LIN {X 0,Y 573.095,Z 768.426,A -85,B 0,C 180,E1 -2257.752,E2 -2257.752} C_VEL
LIN {X 0,Y 573.136,Z 760.652,A -85,B 0,C 180,E1 -2259.172,E2 -2259.172} C_VEL
LIN {X 0,Y 573.27,Z 752.373,A -85,B 0,C 180,E1 -2260.417,E2 -2260.417} C_VEL
LIN {X 0,Y 573.384,Z 742.397,A -85,B 0,C 180,E1 -2261.667,E2 -2261.667} C_VEL
LIN {X 0,Y 573.567,Z 732.195,A -85,B 0,C 180,E1 -2262.741,E2 -2262.741} C_VEL
LIN {X 0,Y 573.742,Z 720.027,A -85,B 0,C 180,E1 -2263.819,E2 -2263.819} C_VEL
LIN {X 0,Y 573.959,Z 706.912,A -85,B 0,C 180,E1 -2264.78,E2 -2264.78} C_VEL
LIN {X 0,Y 574.138,Z 692.882,A -85,B 0,C 180,E1 -2265.622,E2 -2265.622} C_VEL
LIN {X 0,Y 574.337,Z 678.815,A -85,B 0,C 180,E1 -2266.3,E2 -2266.3} C_VEL
LIN {X 0,Y 574.521,Z 664.326,A -85,B 0,C 180,E1 -2266.843,E2 -2266.843} C_VEL
LIN {X 0,Y 574.696,Z 648.452,A -85,B 0,C 180,E1 -2267.274,E2 -2267.274} C_VEL
LIN {X 0,Y 574.79,Z 632.509,A -85,B 0,C 180,E1 -2267.547,E2 -2267.547} C_VEL
LIN {X 0,Y 575.114,Z 478.185,A -85,B 0,C 180,E1 -2269.528,E2 -2269.528} C_VEL
LIN {X 0,Y 574.295,Z 472.988,A -85,B 0,C 180,E1 -2269.647,E2 -2269.647} C_VEL
LIN {X 0,Y 574.659,Z 443.059,A -85,B 0,C 180,E1 -2272.468,E2 -2272.468} C_VEL
LIN {X 0,Y 575.111,Z 413.325,A -85,B 0,C 180,E1 -2275.321,E2 -2275.321} C_VEL
LIN {X 0,Y 575.49,Z 387.313,A -85,B 0,C 180,E1 -2277.839,E2 -2277.839} C_VEL
LIN {X 0,Y 575.461,Z 368.493,A -85,B 0,C 180,E1 -2279.623,E2 -2279.623} C_VEL
LIN {X 0,Y 573.25,Z 359.705,A -85,B 0,C 180,E1 -2280.582,E2 -2280.582} C_VEL
LIN {X 0,Y 573.235,Z 359.704,A -85,B 0,C 180,E1 -2283.52,E2 -2283.52} C_VEL
LIN {X 0,Y 573.175,Z 359.715,A -85,B 0,C 180,E1 -2286.053,E2 -2286.053} C_VEL
LIN {X 0,Y 573.22,Z 359.704,A -85,B 0,C 180,E1 -2288.702,E2 -2288.702} C_VEL
LIN {X 0,Y 573.191,Z 359.706,A -85,B 0,C 180,E1 -2291.459,E2 -2291.459} C_VEL
LIN {X 0,Y 573.203,Z 359.709,A -85,B 0,C 180,E1 -2294.335,E2 -2294.335} C_VEL
LIN {X 0,Y 573.197,Z 359.704,A -85,B 0,C 180,E1 -2297.361,E2 -2297.361} C_VEL
LIN {X 0,Y 573.217,Z 359.708,A -85,B 0,C 180,E1 -2300.391,E2 -2300.391} C_VEL
LIN {X 0,Y 573.201,Z 359.704,A -85,B 0,C 180,E1 -2303.074,E2 -2303.074} C_VEL
LIN {X 0,Y 573.228,Z 359.702,A -85,B 0,C 180,E1 -2305.669,E2 -2305.669} C_VEL
LIN {X 0,Y 573.208,Z 359.712,A -85,B 0,C 180,E1 -2308.183,E2 -2308.183} C_VEL
LIN {X 0,Y 573.205,Z 359.709,A -85,B 0,C 180,E1 -2310.631,E2 -2310.631} C_VEL
LIN {X 0,Y 573.189,Z 359.706,A -85,B 0,C 180,E1 -2313.514,E2 -2313.514} C_VEL
LIN {X 0,Y 573.178,Z 359.713,A -85,B 0,C 180,E1 -2316.132,E2 -2316.132} C_VEL
LIN {X 0,Y 573.201,Z 359.704,A -85,B 0,C 180,E1 -2319.172,E2 -2319.172} C_VEL
LIN {X 0,Y 573.174,Z 359.707,A -85,B 0,C 180,E1 -2321.41,E2 -2321.41} C_VEL
LIN {X 0,Y 573.186,Z 359.715,A -85,B 0,C 180,E1 -2324.351,E2 -2324.351} C_VEL
LIN {X 0,Y 573.173,Z 359.717,A -85,B 0,C 180,E1 -2326.528,E2 -2326.528} C_VEL
LIN {X 0,Y 573.221,Z 359.701,A -85,B 0,C 180,E1 -2329.403,E2 -2329.403} C_VEL
LIN {X 0,Y 573.219,Z 359.708,A -85,B 0,C 180,E1 -2332.249,E2 -2332.249} C_VEL
LIN {X 0,Y 573.262,Z 359.698,A -85,B 0,C 180,E1 -2335.077,E2 -2335.077} C_VEL
LIN {X 0,Y 573.269,Z 359.695,A -85,B 0,C 180,E1 -2337.892,E2 -2337.892} C_VEL
LIN {X 0,Y 573.317,Z 359.697,A -85,B 0,C 180,E1 -2340.703,E2 -2340.703} C_VEL
LIN {X 0,Y 573.283,Z 359.7,A -85,B 0,C 180,E1 -2342.811,E2 -2342.811} C_VEL
LIN {X 0,Y 573.245,Z 359.696,A -85,B 0,C 180,E1 -2345.629,E2 -2345.629} C_VEL
LIN {X 0,Y 573.198,Z 359.7,A -85,B 0,C 180,E1 -2347.751,E2 -2347.751} C_VEL
LIN {X 0,Y 573.23,Z 359.709,A -85,B 0,C 180,E1 -2350.598,E2 -2350.598} C_VEL
LIN {X 0,Y 573.196,Z 359.702,A -85,B 0,C 180,E1 -2353.472,E2 -2353.472} C_VEL
LIN {X 0,Y 573.206,Z 359.701,A -85,B 0,C 180,E1 -2355.649,E2 -2355.649} C_VEL
LIN {X 0,Y 573.207,Z 359.703,A -85,B 0,C 180,E1 -2357.85,E2 -2357.85} C_VEL
LIN {X 0,Y 573.222,Z 359.7,A -85,B 0,C 180,E1 -2360.078,E2 -2360.078} C_VEL
LIN {X 0,Y 573.208,Z 359.704,A -85,B 0,C 180,E1 -2362.339,E2 -2362.339} C_VEL
LIN {X 0,Y 573.193,Z 359.709,A -85,B 0,C 180,E1 -2364.401,E2 -2364.401} C_VEL
LIN {X 0,Y 572.552,Z 359.795,A -85,B 0,C 180,E1 -2364.987,E2 -2364.987} C_VEL
LIN {X 0,Y 569.7,Z 360.151,A -85,B 0,C 180,E1 -2365.939,E2 -2365.939} C_VEL
LIN {X 0,Y 567.274,Z 360.449,A -85,B 0,C 180,E1 -2366.705,E2 -2366.705} C_VEL
LIN {X 0,Y 566.232,Z 360.574,A -85,B 0,C 180,E1 -2367.296,E2 -2367.296} C_VEL
LIN {X 0,Y 566.147,Z 360.583,A -85,B 0,C 180,E1 -2367.496,E2 -2367.496} C_VEL
LIN {X 0,Y 566.158,Z 360.582,A -85,B 0,C 180,E1 -2369.772,E2 -2369.772} C_VEL
LIN {X 0,Y 566.188,Z 360.578,A -85,B 0,C 180,E1 -2372.43,E2 -2372.43} C_VEL
LIN {X 0,Y 566.168,Z 360.588,A -85,B 0,C 180,E1 -2374.99,E2 -2374.99} C_VEL
LIN {X 0,Y 566.184,Z 360.58,A -85,B 0,C 180,E1 -2377.462,E2 -2377.462} C_VEL
LIN {X 0,Y 566.196,Z 360.577,A -85,B 0,C 180,E1 -2380.2,E2 -2380.2} C_VEL
LIN {X 0,Y 566.176,Z 360.586,A -85,B 0,C 180,E1 -2383.057,E2 -2383.057} C_VEL
LIN {X 0,Y 566.185,Z 360.578,A -85,B 0,C 180,E1 -2386.051,E2 -2386.051} C_VEL
LIN {X 0,Y 566.195,Z 360.583,A -85,B 0,C 180,E1 -2389.216,E2 -2389.216} C_VEL
LIN {X 0,Y 566.173,Z 360.581,A -85,B 0,C 180,E1 -2391.637,E2 -2391.637} C_VEL
LIN {X 0,Y 566.138,Z 360.584,A -85,B 0,C 180,E1 -2394.307,E2 -2394.307} C_VEL
LIN {X 0,Y 566.191,Z 360.585,A -85,B 0,C 180,E1 -2396.897,E2 -2396.897} C_VEL
LIN {X 0,Y 566.16,Z 360.588,A -85,B 0,C 180,E1 -2399.407,E2 -2399.407} C_VEL
LIN {X 0,Y 566.169,Z 360.587,A -85,B 0,C 180,E1 -2401.612,E2 -2401.612} C_VEL
LIN {X 0,Y 568.353,Z 366.669,A -85,B 0,C 180,E1 -2401.781,E2 -2401.781} C_VEL
LIN {X 0,Y 567.975,Z 490.989,A -85,B 0,C 180,E1 -2403.409,E2 -2403.409} C_VEL
LIN {X 0,Y 567.841,Z 506.693,A -85,B 0,C 180,E1 -2403.764,E2 -2403.764} C_VEL
LIN {X 0,Y 567.638,Z 522.129,A -85,B 0,C 180,E1 -2404.272,E2 -2404.272} C_VEL
LIN {X 0,Y 567.384,Z 536.347,A -85,B 0,C 180,E1 -2404.89,E2 -2404.89} C_VEL
LIN {X 0,Y 567.131,Z 550.503,A -85,B 0,C 180,E1 -2405.668,E2 -2405.668} C_VEL
LIN {X 0,Y 566.889,Z 563.595,A -85,B 0,C 180,E1 -2406.552,E2 -2406.552} C_VEL
LIN {X 0,Y 566.633,Z 576.205,A -85,B 0,C 180,E1 -2407.581,E2 -2407.581} C_VEL
LIN {X 0,Y 566.434,Z 587.684,A -85,B 0,C 180,E1 -2408.706,E2 -2408.706} C_VEL
LIN {X 0,Y 566.289,Z 597.552,A -85,B 0,C 180,E1 -2409.856,E2 -2409.856} C_VEL
LIN {X 0,Y 566.118,Z 606.994,A -85,B 0,C 180,E1 -2411.17,E2 -2411.17} C_VEL
LIN {X 0,Y 566.04,Z 614.754,A -85,B 0,C 180,E1 -2412.478,E2 -2412.478} C_VEL
LIN {X 0,Y 565.979,Z 621.094,A -85,B 0,C 180,E1 -2413.777,E2 -2413.777} C_VEL
LIN {X 0,Y 565.932,Z 626.848,A -85,B 0,C 180,E1 -2415.252,E2 -2415.252} C_VEL
LIN {X 0,Y 565.884,Z 630.24,A -85,B 0,C 180,E1 -2416.352,E2 -2416.352} C_VEL
LIN {X 0,Y 565.865,Z 633.545,A -85,B 0,C 180,E1 -2417.812,E2 -2417.812} C_VEL
LIN {X 0,Y 565.89,Z 635.583,A -85,B 0,C 180,E1 -2419.264,E2 -2419.264} C_VEL
LIN {X 0,Y 565.822,Z 636.432,A -85,B 0,C 180,E1 -2420.708,E2 -2420.708} C_VEL
LIN {X 0,Y 565.876,Z 636.125,A -85,B 0,C 180,E1 -2422.148,E2 -2422.148} C_VEL
LIN {X 0,Y 565.897,Z 634.669,A -85,B 0,C 180,E1 -2423.583,E2 -2423.583} C_VEL
LIN {X 0,Y 565.855,Z 632.049,A -85,B 0,C 180,E1 -2425.013,E2 -2425.013} C_VEL
LIN {X 0,Y 565.948,Z 628.168,A -85,B 0,C 180,E1 -2426.441,E2 -2426.441} C_VEL
LIN {X 0,Y 565.905,Z 623.007,A -85,B 0,C 180,E1 -2427.865,E2 -2427.865} C_VEL
LIN {X 0,Y 566.023,Z 616.441,A -85,B 0,C 180,E1 -2429.289,E2 -2429.289} C_VEL
LIN {X 0,Y 566.103,Z 609.405,A -85,B 0,C 180,E1 -2430.534,E2 -2430.534} C_VEL
LIN {X 0,Y 566.216,Z 600.993,A -85,B 0,C 180,E1 -2431.778,E2 -2431.778} C_VEL
LIN {X 0,Y 566.393,Z 590.924,A -85,B 0,C 180,E1 -2433.023,E2 -2433.023} C_VEL
LIN {X 0,Y 566.631,Z 580.682,A -85,B 0,C 180,E1 -2434.09,E2 -2434.09} C_VEL
LIN {X 0,Y 566.799,Z 568.495,A -85,B 0,C 180,E1 -2435.158,E2 -2435.158} C_VEL
LIN {X 0,Y 567.019,Z 556.344,A -85,B 0,C 180,E1 -2436.048,E2 -2436.048} C_VEL
LIN {X 0,Y 567.283,Z 543.123,A -85,B 0,C 180,E1 -2436.849,E2 -2436.849} C_VEL
LIN {X 0,Y 567.537,Z 528.88,A -85,B 0,C 180,E1 -2437.543,E2 -2437.543} C_VEL
LIN {X 0,Y 567.774,Z 514.325,A -85,B 0,C 180,E1 -2438.094,E2 -2438.094} C_VEL
LIN {X 0,Y 567.889,Z 499.072,A -85,B 0,C 180,E1 -2438.518,E2 -2438.518} C_VEL
LIN {X 0,Y 567.973,Z 484.215,A -85,B 0,C 180,E1 -2438.786,E2 -2438.786} C_VEL
LIN {X 0,Y 568.274,Z 366.453,A -85,B 0,C 180,E1 -2440.315,E2 -2440.315} C_VEL
LIN {X 0,Y 566.187,Z 360.585,A -85,B 0,C 180,E1 -2440.482,E2 -2440.482} C_VEL
LIN {X 0,Y 566.145,Z 360.593,A -85,B 0,C 180,E1 -2442.912,E2 -2442.912} C_VEL
LIN {X 0,Y 566.155,Z 360.59,A -85,B 0,C 180,E1 -2445.111,E2 -2445.111} C_VEL
LIN {X 0,Y 566.161,Z 360.581,A -85,B 0,C 180,E1 -2448.079,E2 -2448.079} C_VEL
LIN {X 0,Y 566.15,Z 360.584,A -85,B 0,C 180,E1 -2450.339,E2 -2450.339} C_VEL
LIN {X 0,Y 566.131,Z 360.589,A -85,B 0,C 180,E1 -2452.633,E2 -2452.633} C_VEL
LIN {X 0,Y 566.141,Z 360.593,A -85,B 0,C 180,E1 -2455.012,E2 -2455.012} C_VEL
LIN {X 0,Y 566.158,Z 360.587,A -85,B 0,C 180,E1 -2457.341,E2 -2457.341} C_VEL
LIN {X 0,Y 566.143,Z 360.581,A -85,B 0,C 180,E1 -2459.772,E2 -2459.772} C_VEL
LIN {X 0,Y 566.169,Z 360.581,A -85,B 0,C 180,E1 -2462.424,E2 -2462.424} C_VEL
LIN {X 0,Y 566.154,Z 360.589,A -85,B 0,C 180,E1 -2464.985,E2 -2464.985} C_VEL
LIN {X 0,Y 566.184,Z 360.583,A -85,B 0,C 180,E1 -2467.461,E2 -2467.461} C_VEL
LIN {X 0,Y 566.16,Z 360.58,A -85,B 0,C 180,E1 -2470.202,E2 -2470.202} C_VEL
LIN {X 0,Y 566.139,Z 360.592,A -85,B 0,C 180,E1 -2473.059,E2 -2473.059} C_VEL
LIN {X 0,Y 566.147,Z 360.583,A -85,B 0,C 180,E1 -2476.053,E2 -2476.053} C_VEL
LIN {X 0,Y 566.165,Z 360.59,A -85,B 0,C 180,E1 -2479.218,E2 -2479.218} C_VEL
LIN {X 0,Y 566.138,Z 360.587,A -85,B 0,C 180,E1 -2481.633,E2 -2481.633} C_VEL
LIN {X 0,Y 566.133,Z 360.584,A -85,B 0,C 180,E1 -2484.305,E2 -2484.305} C_VEL
LIN {X 0,Y 566.154,Z 360.584,A -85,B 0,C 180,E1 -2486.893,E2 -2486.893} C_VEL
LIN {X 0,Y 566.141,Z 360.591,A -85,B 0,C 180,E1 -2489.405,E2 -2489.405} C_VEL
LIN {X 0,Y 566.138,Z 360.586,A -85,B 0,C 180,E1 -2491.853,E2 -2491.853} C_VEL
LIN {X 0,Y 566.158,Z 360.581,A -85,B 0,C 180,E1 -2494.248,E2 -2494.248} C_VEL
LIN {X 0,Y 566.151,Z 360.592,A -85,B 0,C 180,E1 -2497.367,E2 -2497.367} C_VEL
LIN {X 0,Y 566.189,Z 360.582,A -85,B 0,C 180,E1 -2499.662,E2 -2499.662} C_VEL
LIN {X 0,Y 566.156,Z 360.583,A -85,B 0,C 180,E1 -2501.92,E2 -2501.92} C_VEL
LIN {X 0,Y 566.172,Z 360.582,A -85,B 0,C 180,E1 -2504.89,E2 -2504.89} C_VEL
LIN {X 0,Y 566.165,Z 360.578,A -85,B 0,C 180,E1 -2507.817,E2 -2507.817} C_VEL
LIN {X 0,Y 566.126,Z 360.582,A -85,B 0,C 180,E1 -2509.991,E2 -2509.991} C_VEL
LIN {X 0,Y 566.168,Z 360.579,A -85,B 0,C 180,E1 -2512.152,E2 -2512.152} C_VEL
LIN {X 0,Y 566.255,Z 360.572,A -85,B 0,C 180,E1 -2515.016,E2 -2515.016} C_VEL
LIN {X 0,Y 566.248,Z 360.573,A -85,B 0,C 180,E1 -2517.866,E2 -2517.866} C_VEL
LIN {X 0,Y 566.255,Z 360.572,A -85,B 0,C 180,E1 -2520,E2 -2520} C_VEL
LIN {X 0,Y 566.233,Z 360.572,A -85,B 0,C 180,E1 -2522.846,E2 -2522.846} C_VEL
LIN {X 0,Y 566.223,Z 360.581,A -85,B 0,C 180,E1 -2525.698,E2 -2525.698} C_VEL
LIN {X 0,Y 566.165,Z 360.579,A -85,B 0,C 180,E1 -2528.566,E2 -2528.566} C_VEL
LIN {X 0,Y 566.226,Z 360.58,A -85,B 0,C 180,E1 -2531.454,E2 -2531.454} C_VEL
LIN {X 0,Y 566.191,Z 360.576,A -85,B 0,C 180,E1 -2534.494,E2 -2534.494} C_VEL
LIN {X 0,Y 566.146,Z 360.588,A -85,B 0,C 180,E1 -2537.333,E2 -2537.333} C_VEL
LIN {X 0,Y 566.163,Z 360.588,A -85,B 0,C 180,E1 -2539.582,E2 -2539.582} C_VEL
LIN {X 0,Y 566.135,Z 360.59,A -85,B 0,C 180,E1 -2541.865,E2 -2541.865} C_VEL
LIN {X 0,Y 566.183,Z 360.579,A -85,B 0,C 180,E1 -2544.963,E2 -2544.963} C_VEL
LIN {X 0,Y 566.148,Z 360.586,A -85,B 0,C 180,E1 -2547.342,E2 -2547.342} C_VEL
LIN {X 0,Y 566.149,Z 360.592,A -85,B 0,C 180,E1 -2549.772,E2 -2549.772} C_VEL
LIN {X 0,Y 566.166,Z 360.58,A -85,B 0,C 180,E1 -2552.426,E2 -2552.426} C_VEL
LIN {X 0,Y 566.153,Z 360.581,A -85,B 0,C 180,E1 -2554.987,E2 -2554.987} C_VEL
LIN {X 0,Y 566.173,Z 360.584,A -85,B 0,C 180,E1 -2557.463,E2 -2557.463} C_VEL
LIN {X 0,Y 566.195,Z 360.581,A -85,B 0,C 180,E1 -2560.2,E2 -2560.2} C_VEL
LIN {X 0,Y 566.134,Z 360.584,A -85,B 0,C 180,E1 -2563.06,E2 -2563.06} C_VEL
LIN {X 0,Y 566.147,Z 360.59,A -85,B 0,C 180,E1 -2566.054,E2 -2566.054} C_VEL
LIN {X 0,Y 566.132,Z 360.582,A -85,B 0,C 180,E1 -2568.858,E2 -2568.858} C_VEL
LIN {X 0,Y 566.167,Z 360.586,A -85,B 0,C 180,E1 -2571.636,E2 -2571.636} C_VEL
LIN {X 0,Y 566.131,Z 360.59,A -85,B 0,C 180,E1 -2574.306,E2 -2574.306} C_VEL
LIN {X 0,Y 566.158,Z 360.584,A -85,B 0,C 180,E1 -2576.894,E2 -2576.894} C_VEL
LIN {X 0,Y 566.183,Z 360.71,A -85,B 0,C 180,E1 -2579.186,E2 -2579.186} C_VEL
LIN {X 0,Y 568.608,Z 369.797,A -85,B 0,C 180,E1 -2580.186,E2 -2580.186} C_VEL
LIN {X 0,Y 568.694,Z 381.61,A -85,B 0,C 180,E1 -2581.333,E2 -2581.333} C_VEL
LIN {X 0,Y 568.501,Z 408.247,A -85,B 0,C 180,E1 -2583.871,E2 -2583.871} C_VEL
LIN {X 0,Y 568.018,Z 435.853,A -85,B 0,C 180,E1 -2586.554,E2 -2586.554} C_VEL
LIN {X 0,Y 567.548,Z 464.858,A -85,B 0,C 180,E1 -2589.334,E2 -2589.334} C_VEL
LIN {X 0,Y 567.46,Z 473.303,A -85,B 0,C 180,E1 -2590.133,E2 -2590.133} C_VEL
LIN {X 0,Y 568.498,Z 480.342,A -85,B 0,C 180,E1 -2590.264,E2 -2590.264} C_VEL
LIN {X 0,Y 567.995,Z 640.714,A -85,B 0,C 180,E1 -2592.36,E2 -2592.36} C_VEL
LIN {X 0,Y 567.839,Z 656.165,A -85,B 0,C 180,E1 -2592.705,E2 -2592.705} C_VEL
LIN {X 0,Y 567.658,Z 670.801,A -85,B 0,C 180,E1 -2593.178,E2 -2593.178} C_VEL
LIN {X 0,Y 567.491,Z 683.806,A -85,B 0,C 180,E1 -2593.728,E2 -2593.728} C_VEL
LIN {X 0,Y 567.175,Z 697.681,A -85,B 0,C 180,E1 -2594.457,E2 -2594.457} C_VEL
LIN {X 0,Y 566.935,Z 711.501,A -85,B 0,C 180,E1 -2595.358,E2 -2595.358} C_VEL
LIN {X 0,Y 566.672,Z 724.291,A -85,B 0,C 180,E1 -2596.371,E2 -2596.371} C_VEL
LIN {X 0,Y 566.491,Z 735.749,A -85,B 0,C 180,E1 -2597.461,E2 -2597.461} C_VEL
LIN {X 0,Y 566.268,Z 746.312,A -85,B 0,C 180,E1 -2598.659,E2 -2598.659} C_VEL
LIN {X 0,Y 566.208,Z 754.857,A -85,B 0,C 180,E1 -2599.812,E2 -2599.812} C_VEL
LIN {X 0,Y 566.057,Z 762.733,A -85,B 0,C 180,E1 -2601.072,E2 -2601.072} C_VEL
LIN {X 0,Y 565.997,Z 770.089,A -85,B 0,C 180,E1 -2602.508,E2 -2602.508} C_VEL
LIN {X 0,Y 565.956,Z 775.922,A -85,B 0,C 180,E1 -2603.941,E2 -2603.941} C_VEL
LIN {X 0,Y 565.866,Z 779.385,A -85,B 0,C 180,E1 -2605.012,E2 -2605.012} C_VEL
LIN {X 0,Y 565.909,Z 782.889,A -85,B 0,C 180,E1 -2606.44,E2 -2606.44} C_VEL
LIN {X 0,Y 565.836,Z 785.192,A -85,B 0,C 180,E1 -2607.864,E2 -2607.864} C_VEL
LIN {X 0,Y 565.838,Z 786.349,A -85,B 0,C 180,E1 -2609.288,E2 -2609.288} C_VEL
LIN {X 0,Y 565.838,Z 786.349,A -85,B 0,C 180,E1 -2610.711,E2 -2610.711} C_VEL
LIN {X 0,Y 565.836,Z 785.191,A -85,B 0,C 180,E1 -2612.135,E2 -2612.135} C_VEL
LIN {X 0,Y 565.909,Z 782.888,A -85,B 0,C 180,E1 -2613.56,E2 -2613.56} C_VEL
LIN {X 0,Y 565.866,Z 779.387,A -85,B 0,C 180,E1 -2614.987,E2 -2614.987} C_VEL
LIN {X 0,Y 565.956,Z 775.926,A -85,B 0,C 180,E1 -2616.059,E2 -2616.059} C_VEL
LIN {X 0,Y 565.999,Z 770.09,A -85,B 0,C 180,E1 -2617.491,E2 -2617.491} C_VEL
LIN {X 0,Y 566.057,Z 762.733,A -85,B 0,C 180,E1 -2618.928,E2 -2618.928} C_VEL
LIN {X 0,Y 566.208,Z 754.86,A -85,B 0,C 180,E1 -2620.187,E2 -2620.187} C_VEL
LIN {X 0,Y 566.307,Z 745.395,A -85,B 0,C 180,E1 -2621.452,E2 -2621.452} C_VEL
LIN {X 0,Y 566.491,Z 735.754,A -85,B 0,C 180,E1 -2622.539,E2 -2622.539} C_VEL
LIN {X 0,Y 566.671,Z 724.301,A -85,B 0,C 180,E1 -2623.629,E2 -2623.629} C_VEL
LIN {X 0,Y 566.926,Z 711.684,A -85,B 0,C 180,E1 -2624.63,E2 -2624.63} C_VEL
LIN {X 0,Y 567.15,Z 699.255,A -85,B 0,C 180,E1 -2625.451,E2 -2625.451} C_VEL
LIN {X 0,Y 567.418,Z 685.782,A -85,B 0,C 180,E1 -2626.181,E2 -2626.181} C_VEL
LIN {X 0,Y 567.606,Z 672.065,A -85,B 0,C 180,E1 -2626.777,E2 -2626.777} C_VEL
LIN {X 0,Y 567.845,Z 656.743,A -85,B 0,C 180,E1 -2627.279,E2 -2627.279} C_VEL
LIN {X 0,Y 567.978,Z 641.336,A -85,B 0,C 180,E1 -2627.629,E2 -2627.629} C_VEL
LIN {X 0,Y 568.451,Z 479.257,A -85,B 0,C 180,E1 -2629.752,E2 -2629.752} C_VEL
LIN {X 0,Y 567.456,Z 473.137,A -85,B 0,C 180,E1 -2629.879,E2 -2629.879} C_VEL
LIN {X 0,Y 567.9,Z 443.059,A -85,B 0,C 180,E1 -2632.75,E2 -2632.75} C_VEL
LIN {X 0,Y 568.442,Z 413.325,A -85,B 0,C 180,E1 -2635.64,E2 -2635.64} C_VEL
LIN {X 0,Y 568.649,Z 384.809,A -85,B 0,C 180,E1 -2638.347,E2 -2638.347} C_VEL
LIN {X 0,Y 568.585,Z 369.664,A -85,B 0,C 180,E1 -2639.805,E2 -2639.805} C_VEL
LIN {X 0,Y 566.189,Z 360.584,A -85,B 0,C 180,E1 -2640.814,E2 -2640.814} C_VEL
LIN {X 0,Y 566.188,Z 360.58,A -85,B 0,C 180,E1 -2643.103,E2 -2643.103} C_VEL
LIN {X 0,Y 566.129,Z 360.59,A -85,B 0,C 180,E1 -2645.693,E2 -2645.693} C_VEL
LIN {X 0,Y 566.191,Z 360.581,A -85,B 0,C 180,E1 -2648.556,E2 -2648.556} C_VEL
LIN {X 0,Y 566.145,Z 360.583,A -85,B 0,C 180,E1 -2651.141,E2 -2651.141} C_VEL
LIN {X 0,Y 566.144,Z 360.59,A -85,B 0,C 180,E1 -2653.946,E2 -2653.946} C_VEL
LIN {X 0,Y 566.135,Z 360.584,A -85,B 0,C 180,E1 -2657.088,E2 -2657.088} C_VEL
LIN {X 0,Y 566.194,Z 360.584,A -85,B 0,C 180,E1 -2660.315,E2 -2660.315} C_VEL
LIN {X 0,Y 566.171,Z 360.584,A -85,B 0,C 180,E1 -2662.601,E2 -2662.601} C_VEL
LIN {X 0,Y 566.166,Z 360.581,A -85,B 0,C 180,E1 -2665.179,E2 -2665.179} C_VEL
LIN {X 0,Y 566.193,Z 360.579,A -85,B 0,C 180,E1 -2667.741,E2 -2667.741} C_VEL
LIN {X 0,Y 566.143,Z 360.593,A -85,B 0,C 180,E1 -2670.336,E2 -2670.336} C_VEL
LIN {X 0,Y 566.164,Z 360.581,A -85,B 0,C 180,E1 -2673.456,E2 -2673.456} C_VEL
LIN {X 0,Y 566.14,Z 360.586,A -85,B 0,C 180,E1 -2675.817,E2 -2675.817} C_VEL
LIN {X 0,Y 566.166,Z 360.582,A -85,B 0,C 180,E1 -2678.901,E2 -2678.901} C_VEL
LIN {X 0,Y 566.151,Z 360.583,A -85,B 0,C 180,E1 -2681.171,E2 -2681.171} C_VEL
LIN {X 0,Y 566.153,Z 360.587,A -85,B 0,C 180,E1 -2684.151,E2 -2684.151} C_VEL
LIN {X 0,Y 566.139,Z 360.592,A -85,B 0,C 180,E1 -2686.358,E2 -2686.358} C_VEL
LIN {X 0,Y 566.2,Z 360.576,A -85,B 0,C 180,E1 -2689.27,E2 -2689.27} C_VEL
LIN {X 0,Y 566.182,Z 360.583,A -85,B 0,C 180,E1 -2692.152,E2 -2692.152} C_VEL
LIN {X 0,Y 566.238,Z 360.574,A -85,B 0,C 180,E1 -2695.016,E2 -2695.016} C_VEL
LIN {X 0,Y 566.242,Z 360.57,A -85,B 0,C 180,E1 -2697.866,E2 -2697.866} C_VEL
LIN {X 0,Y 566.286,Z 360.572,A -85,B 0,C 180,E1 -2700.711,E2 -2700.711} C_VEL
LIN {X 0,Y 566.247,Z 360.576,A -85,B 0,C 180,E1 -2702.846,E2 -2702.846} C_VEL
LIN {X 0,Y 566.215,Z 360.571,A -85,B 0,C 180,E1 -2705.699,E2 -2705.699} C_VEL
LIN {X 0,Y 566.169,Z 360.576,A -85,B 0,C 180,E1 -2707.848,E2 -2707.848} C_VEL
LIN {X 0,Y 566.207,Z 360.584,A -85,B 0,C 180,E1 -2710.731,E2 -2710.731} C_VEL
LIN {X 0,Y 566.162,Z 360.577,A -85,B 0,C 180,E1 -2713.642,E2 -2713.642} C_VEL
LIN {X 0,Y 566.192,Z 360.583,A -85,B 0,C 180,E1 -2716.589,E2 -2716.589} C_VEL
LIN {X 0,Y 566.186,Z 360.576,A -85,B 0,C 180,E1 -2719.582,E2 -2719.582} C_VEL
LIN {X 0,Y 566.172,Z 360.577,A -85,B 0,C 180,E1 -2721.864,E2 -2721.864} C_VEL
LIN {X 0,Y 566.165,Z 360.585,A -85,B 0,C 180,E1 -2725.022,E2 -2725.022} C_VEL
LIN {X 0,Y 566.147,Z 360.583,A -85,B 0,C 180,E1 -2727.496,E2 -2727.496} C_VEL
LIN {X 0,Y 565.48,Z 360.666,A -85,B 0,C 180,E1 -2728.09,E2 -2728.09} C_VEL
LIN {X 0,Y 562.624,Z 361.029,A -85,B 0,C 180,E1 -2729.054,E2 -2729.054} C_VEL
LIN {X 0,Y 560.217,Z 361.325,A -85,B 0,C 180,E1 -2729.83,E2 -2729.83} C_VEL
LIN {X 0,Y 559.194,Z 361.453,A -85,B 0,C 180,E1 -2730.429,E2 -2730.429} C_VEL
LIN {X 0,Y 559.116,Z 361.46,A -85,B 0,C 180,E1 -2730.631,E2 -2730.631} C_VEL
LIN {X 0,Y 559.138,Z 361.46,A -85,B 0,C 180,E1 -2732.717,E2 -2732.717} C_VEL
LIN {X 0,Y 559.116,Z 361.461,A -85,B 0,C 180,E1 -2735.325,E2 -2735.325} C_VEL
LIN {X 0,Y 559.118,Z 361.458,A -85,B 0,C 180,E1 -2738.019,E2 -2738.019} C_VEL
LIN {X 0,Y 559.144,Z 361.462,A -85,B 0,C 180,E1 -2740.814,E2 -2740.814} C_VEL
LIN {X 0,Y 559.101,Z 361.459,A -85,B 0,C 180,E1 -2743.738,E2 -2743.738} C_VEL
LIN {X 0,Y 559.128,Z 361.458,A -85,B 0,C 180,E1 -2746.267,E2 -2746.267} C_VEL
LIN {X 0,Y 559.147,Z 361.461,A -85,B 0,C 180,E1 -2749.188,E2 -2749.188} C_VEL
LIN {X 0,Y 559.122,Z 361.457,A -85,B 0,C 180,E1 -2751.983,E2 -2751.983} C_VEL
LIN {X 0,Y 559.119,Z 361.463,A -85,B 0,C 180,E1 -2754.79,E2 -2754.79} C_VEL
LIN {X 0,Y 559.145,Z 361.461,A -85,B 0,C 180,E1 -2757.367,E2 -2757.367} C_VEL
LIN {X 0,Y 559.109,Z 361.462,A -85,B 0,C 180,E1 -2760.15,E2 -2760.15} C_VEL
LIN {X 0,Y 559.117,Z 361.527,A -85,B 0,C 180,E1 -2761.379,E2 -2761.379} C_VEL
LIN {X 0,Y 561.634,Z 368.25,A -85,B 0,C 180,E1 -2761.562,E2 -2761.562} C_VEL
LIN {X 0,Y 561.219,Z 491.044,A -85,B 0,C 180,E1 -2763.191,E2 -2763.191} C_VEL
LIN {X 0,Y 561.067,Z 506.667,A -85,B 0,C 180,E1 -2763.548,E2 -2763.548} C_VEL
LIN {X 0,Y 560.824,Z 522.232,A -85,B 0,C 180,E1 -2764.067,E2 -2764.067} C_VEL
LIN {X 0,Y 560.536,Z 536.555,A -85,B 0,C 180,E1 -2764.698,E2 -2764.698} C_VEL
LIN {X 0,Y 560.252,Z 550.083,A -85,B 0,C 180,E1 -2765.448,E2 -2765.448} C_VEL
LIN {X 0,Y 559.968,Z 563.716,A -85,B 0,C 180,E1 -2766.378,E2 -2766.378} C_VEL
LIN {X 0,Y 559.697,Z 575.924,A -85,B 0,C 180,E1 -2767.385,E2 -2767.385} C_VEL
LIN {X 0,Y 559.507,Z 586.793,A -85,B 0,C 180,E1 -2768.455,E2 -2768.455} C_VEL
LIN {X 0,Y 559.249,Z 598.086,A -85,B 0,C 180,E1 -2769.783,E2 -2769.783} C_VEL
LIN {X 0,Y 559.077,Z 607.431,A -85,B 0,C 180,E1 -2771.114,E2 -2771.114} C_VEL
LIN {X 0,Y 558.972,Z 615.134,A -85,B 0,C 180,E1 -2772.438,E2 -2772.438} C_VEL
LIN {X 0,Y 558.868,Z 622.222,A -85,B 0,C 180,E1 -2773.94,E2 -2773.94} C_VEL
LIN {X 0,Y 558.855,Z 627.719,A -85,B 0,C 180,E1 -2775.434,E2 -2775.434} C_VEL
LIN {X 0,Y 558.751,Z 631.776,A -85,B 0,C 180,E1 -2776.915,E2 -2776.915} C_VEL
LIN {X 0,Y 558.774,Z 634.539,A -85,B 0,C 180,E1 -2778.391,E2 -2778.391} C_VEL
LIN {X 0,Y 558.774,Z 636.079,A -85,B 0,C 180,E1 -2779.859,E2 -2779.859} C_VEL
LIN {X 0,Y 558.762,Z 636.447,A -85,B 0,C 180,E1 -2781.319,E2 -2781.319} C_VEL
LIN {X 0,Y 558.795,Z 635.665,A -85,B 0,C 180,E1 -2782.775,E2 -2782.775} C_VEL
LIN {X 0,Y 558.83,Z 633.721,A -85,B 0,C 180,E1 -2784.226,E2 -2784.226} C_VEL
LIN {X 0,Y 558.809,Z 630.549,A -85,B 0,C 180,E1 -2785.673,E2 -2785.673} C_VEL
LIN {X 0,Y 558.819,Z 626.144,A -85,B 0,C 180,E1 -2787.117,E2 -2787.117} C_VEL
LIN {X 0,Y 558.85,Z 620.417,A -85,B 0,C 180,E1 -2788.559,E2 -2788.559} C_VEL
LIN {X 0,Y 559.013,Z 613.212,A -85,B 0,C 180,E1 -2790,E2 -2790} C_VEL
LIN {X 0,Y 559.174,Z 604.329,A -85,B 0,C 180,E1 -2791.441,E2 -2791.441} C_VEL
LIN {X 0,Y 559.293,Z 594.924,A -85,B 0,C 180,E1 -2792.701,E2 -2792.701} C_VEL
LIN {X 0,Y 559.51,Z 585.382,A -85,B 0,C 180,E1 -2793.781,E2 -2793.781} C_VEL
LIN {X 0,Y 559.74,Z 574.116,A -85,B 0,C 180,E1 -2794.862,E2 -2794.862} C_VEL
LIN {X 0,Y 559.983,Z 561.785,A -85,B 0,C 180,E1 -2795.853,E2 -2795.853} C_VEL
LIN {X 0,Y 560.298,Z 548.188,A -85,B 0,C 180,E1 -2796.753,E2 -2796.753} C_VEL
LIN {X 0,Y 560.559,Z 535.225,A -85,B 0,C 180,E1 -2797.456,E2 -2797.456} C_VEL
LIN {X 0,Y 560.838,Z 520.072,A -85,B 0,C 180,E1 -2798.104,E2 -2798.104} C_VEL
LIN {X 0,Y 561.044,Z 505.334,A -85,B 0,C 180,E1 -2798.577,E2 -2798.577} C_VEL
LIN {X 0,Y 561.198,Z 490.077,A -85,B 0,C 180,E1 -2798.915,E2 -2798.915} C_VEL
LIN {X 0,Y 561.55,Z 368.078,A -85,B 0,C 180,E1 -2800.533,E2 -2800.533} C_VEL
LIN {X 0,Y 559.201,Z 361.62,A -85,B 0,C 180,E1 -2800.706,E2 -2800.706} C_VEL
LIN {X 0,Y 559.12,Z 361.467,A -85,B 0,C 180,E1 -2803.077,E2 -2803.077} C_VEL
LIN {X 0,Y 559.13,Z 361.457,A -85,B 0,C 180,E1 -2806.053,E2 -2806.053} C_VEL
LIN {X 0,Y 559.141,Z 361.465,A -85,B 0,C 180,E1 -2809.075,E2 -2809.075} C_VEL
LIN {X 0,Y 559.129,Z 361.46,A -85,B 0,C 180,E1 -2811.542,E2 -2811.542} C_VEL
LIN {X 0,Y 559.086,Z 361.465,A -85,B 0,C 180,E1 -2814.508,E2 -2814.508} C_VEL
LIN {X 0,Y 559.112,Z 361.467,A -85,B 0,C 180,E1 -2816.905,E2 -2816.905} C_VEL
LIN {X 0,Y 559.093,Z 361.458,A -85,B 0,C 180,E1 -2819.847,E2 -2819.847} C_VEL
LIN {X 0,Y 559.131,Z 361.461,A -85,B 0,C 180,E1 -2822.716,E2 -2822.716} C_VEL
LIN {X 0,Y 559.108,Z 361.466,A -85,B 0,C 180,E1 -2825.325,E2 -2825.325} C_VEL
LIN {X 0,Y 559.113,Z 361.459,A -85,B 0,C 180,E1 -2828.018,E2 -2828.018} C_VEL
LIN {X 0,Y 559.098,Z 361.464,A -85,B 0,C 180,E1 -2830.817,E2 -2830.817} C_VEL
LIN {X 0,Y 559.088,Z 361.463,A -85,B 0,C 180,E1 -2833.738,E2 -2833.738} C_VEL
LIN {X 0,Y 559.093,Z 361.461,A -85,B 0,C 180,E1 -2836.261,E2 -2836.261} C_VEL
LIN {X 0,Y 559.117,Z 361.467,A -85,B 0,C 180,E1 -2839.184,E2 -2839.184} C_VEL
LIN {X 0,Y 559.126,Z 361.466,A -85,B 0,C 180,E1 -2841.197,E2 -2841.197} C_VEL
LIN {X 0,Y 559.108,Z 361.462,A -85,B 0,C 180,E1 -2843.787,E2 -2843.787} C_VEL
LIN {X 0,Y 559.116,Z 361.457,A -85,B 0,C 180,E1 -2846.422,E2 -2846.422} C_VEL
LIN {X 0,Y 559.127,Z 361.462,A -85,B 0,C 180,E1 -2848.979,E2 -2848.979} C_VEL
LIN {X 0,Y 559.099,Z 361.465,A -85,B 0,C 180,E1 -2851.63,E2 -2851.63} C_VEL
LIN {X 0,Y 559.105,Z 361.462,A -85,B 0,C 180,E1 -2853.899,E2 -2853.899} C_VEL
LIN {X 0,Y 559.101,Z 361.464,A -85,B 0,C 180,E1 -2857.065,E2 -2857.065} C_VEL
LIN {X 0,Y 559.161,Z 361.462,A -85,B 0,C 180,E1 -2859.395,E2 -2859.395} C_VEL
LIN {X 0,Y 559.107,Z 361.464,A -85,B 0,C 180,E1 -2861.684,E2 -2861.684} C_VEL
LIN {X 0,Y 559.13,Z 361.459,A -85,B 0,C 180,E1 -2863.947,E2 -2863.947} C_VEL
LIN {X 0,Y 559.133,Z 361.455,A -85,B 0,C 180,E1 -2866.183,E2 -2866.183} C_VEL
LIN {X 0,Y 559.167,Z 361.45,A -85,B 0,C 180,E1 -2869.133,E2 -2869.133} C_VEL
LIN {X 0,Y 559.123,Z 361.458,A -85,B 0,C 180,E1 -2872.052,E2 -2872.052} C_VEL
LIN {X 0,Y 559.228,Z 361.447,A -85,B 0,C 180,E1 -2874.953,E2 -2874.953} C_VEL
LIN {X 0,Y 559.221,Z 361.448,A -85,B 0,C 180,E1 -2877.839,E2 -2877.839} C_VEL
LIN {X 0,Y 559.226,Z 361.447,A -85,B 0,C 180,E1 -2880,E2 -2880} C_VEL
LIN {X 0,Y 559.203,Z 361.448,A -85,B 0,C 180,E1 -2882.881,E2 -2882.881} C_VEL
LIN {X 0,Y 559.19,Z 361.456,A -85,B 0,C 180,E1 -2885.77,E2 -2885.77} C_VEL
LIN {X 0,Y 559.132,Z 361.455,A -85,B 0,C 180,E1 -2888.675,E2 -2888.675} C_VEL
LIN {X 0,Y 559.183,Z 361.46,A -85,B 0,C 180,E1 -2891.601,E2 -2891.601} C_VEL
LIN {X 0,Y 559.141,Z 361.454,A -85,B 0,C 180,E1 -2894.576,E2 -2894.576} C_VEL
LIN {X 0,Y 559.101,Z 361.469,A -85,B 0,C 180,E1 -2897.559,E2 -2897.559} C_VEL
LIN {X 0,Y 559.126,Z 361.465,A -85,B 0,C 180,E1 -2899.839,E2 -2899.839} C_VEL
LIN {X 0,Y 559.091,Z 361.464,A -85,B 0,C 180,E1 -2902.155,E2 -2902.155} C_VEL
LIN {X 0,Y 559.128,Z 361.459,A -85,B 0,C 180,E1 -2905.178,E2 -2905.178} C_VEL
LIN {X 0,Y 559.09,Z 361.471,A -85,B 0,C 180,E1 -2907.717,E2 -2907.717} C_VEL
LIN {X 0,Y 559.12,Z 361.462,A -85,B 0,C 180,E1 -2910.185,E2 -2910.185} C_VEL
LIN {X 0,Y 559.124,Z 361.456,A -85,B 0,C 180,E1 -2912.717,E2 -2912.717} C_VEL
LIN {X 0,Y 559.105,Z 361.462,A -85,B 0,C 180,E1 -2915.326,E2 -2915.326} C_VEL
LIN {X 0,Y 559.106,Z 361.465,A -85,B 0,C 180,E1 -2918.02,E2 -2918.02} C_VEL
LIN {X 0,Y 559.117,Z 361.459,A -85,B 0,C 180,E1 -2920.816,E2 -2920.816} C_VEL
LIN {X 0,Y 559.085,Z 361.47,A -85,B 0,C 180,E1 -2923.739,E2 -2923.739} C_VEL
LIN {X 0,Y 559.099,Z 361.465,A -85,B 0,C 180,E1 -2926.263,E2 -2926.263} C_VEL
LIN {X 0,Y 559.09,Z 361.459,A -85,B 0,C 180,E1 -2928.958,E2 -2928.958} C_VEL
LIN {X 0,Y 559.161,Z 361.454,A -85,B 0,C 180,E1 -2931.193,E2 -2931.193} C_VEL
LIN {X 0,Y 559.106,Z 361.468,A -85,B 0,C 180,E1 -2933.787,E2 -2933.787} C_VEL
LIN {X 0,Y 559.132,Z 361.462,A -85,B 0,C 180,E1 -2936.424,E2 -2936.424} C_VEL
LIN {X 0,Y 559.142,Z 361.498,A -85,B 0,C 180,E1 -2938.935,E2 -2938.935} C_VEL
LIN {X 0,Y 561.856,Z 371.79,A -85,B 0,C 180,E1 -2940.081,E2 -2940.081} C_VEL
LIN {X 0,Y 561.91,Z 383.47,A -85,B 0,C 180,E1 -2941.228,E2 -2941.228} C_VEL
LIN {X 0,Y 561.647,Z 410.435,A -85,B 0,C 180,E1 -2943.827,E2 -2943.827} C_VEL
LIN {X 0,Y 561.283,Z 435.475,A -85,B 0,C 180,E1 -2946.218,E2 -2946.218} C_VEL
LIN {X 0,Y 560.753,Z 462.876,A -85,B 0,C 180,E1 -2948.88,E2 -2948.88} C_VEL
LIN {X 0,Y 560.613,Z 473.15,A -85,B 0,C 180,E1 -2949.869,E2 -2949.869} C_VEL
LIN {X 0,Y 561.838,Z 481.266,A -85,B 0,C 180,E1 -2950.032,E2 -2950.032} C_VEL
LIN {X 0,Y 561.227,Z 640.56,A -85,B 0,C 180,E1 -2952.138,E2 -2952.138} C_VEL
LIN {X 0,Y 561.071,Z 656.226,A -85,B 0,C 180,E1 -2952.492,E2 -2952.492} C_VEL
LIN {X 0,Y 560.853,Z 670.802,A -85,B 0,C 180,E1 -2952.968,E2 -2952.968} C_VEL
LIN {X 0,Y 560.638,Z 683.807,A -85,B 0,C 180,E1 -2953.524,E2 -2953.524} C_VEL
LIN {X 0,Y 560.316,Z 697.681,A -85,B 0,C 180,E1 -2954.262,E2 -2954.262} C_VEL
LIN {X 0,Y 560.024,Z 711.502,A -85,B 0,C 180,E1 -2955.173,E2 -2955.173} C_VEL
LIN {X 0,Y 559.722,Z 724.292,A -85,B 0,C 180,E1 -2956.198,E2 -2956.198} C_VEL
LIN {X 0,Y 559.516,Z 735.75,A -85,B 0,C 180,E1 -2957.302,E2 -2957.302} C_VEL
LIN {X 0,Y 559.304,Z 745.39,A -85,B 0,C 180,E1 -2958.402,E2 -2958.402} C_VEL
LIN {X 0,Y 559.168,Z 754.856,A -85,B 0,C 180,E1 -2959.682,E2 -2959.682} C_VEL
LIN {X 0,Y 559.003,Z 762.734,A -85,B 0,C 180,E1 -2960.958,E2 -2960.958} C_VEL
LIN {X 0,Y 558.92,Z 770.089,A -85,B 0,C 180,E1 -2962.413,E2 -2962.413} C_VEL
LIN {X 0,Y 558.858,Z 775.922,A -85,B 0,C 180,E1 -2963.864,E2 -2963.864} C_VEL
LIN {X 0,Y 558.787,Z 779.385,A -85,B 0,C 180,E1 -2964.949,E2 -2964.949} C_VEL
LIN {X 0,Y 558.818,Z 782.889,A -85,B 0,C 180,E1 -2966.395,E2 -2966.395} C_VEL
LIN {X 0,Y 558.742,Z 785.191,A -85,B 0,C 180,E1 -2967.837,E2 -2967.837} C_VEL
LIN {X 0,Y 558.739,Z 786.349,A -85,B 0,C 180,E1 -2969.279,E2 -2969.279} C_VEL
LIN {X 0,Y 558.739,Z 786.348,A -85,B 0,C 180,E1 -2970.72,E2 -2970.72} C_VEL
LIN {X 0,Y 558.742,Z 785.19,A -85,B 0,C 180,E1 -2972.162,E2 -2972.162} C_VEL
LIN {X 0,Y 558.818,Z 782.887,A -85,B 0,C 180,E1 -2973.605,E2 -2973.605} C_VEL
LIN {X 0,Y 558.787,Z 779.387,A -85,B 0,C 180,E1 -2975.05,E2 -2975.05} C_VEL
LIN {X 0,Y 558.842,Z 774.61,A -85,B 0,C 180,E1 -2976.498,E2 -2976.498} C_VEL
LIN {X 0,Y 558.951,Z 768.425,A -85,B 0,C 180,E1 -2977.95,E2 -2977.95} C_VEL
LIN {X 0,Y 559.005,Z 760.65,A -85,B 0,C 180,E1 -2979.406,E2 -2979.406} C_VEL
LIN {X 0,Y 559.216,Z 752.372,A -85,B 0,C 180,E1 -2980.682,E2 -2980.682} C_VEL
LIN {X 0,Y 559.361,Z 742.396,A -85,B 0,C 180,E1 -2981.964,E2 -2981.964} C_VEL
LIN {X 0,Y 559.595,Z 732.193,A -85,B 0,C 180,E1 -2983.065,E2 -2983.065} C_VEL
LIN {X 0,Y 559.86,Z 720.027,A -85,B 0,C 180,E1 -2984.169,E2 -2984.169} C_VEL
LIN {X 0,Y 560.128,Z 707.699,A -85,B 0,C 180,E1 -2985.099,E2 -2985.099} C_VEL
LIN {X 0,Y 560.357,Z 694.524,A -85,B 0,C 180,E1 -2985.923,E2 -2985.923} C_VEL
LIN {X 0,Y 560.669,Z 679.844,A -85,B 0,C 180,E1 -2986.662,E2 -2986.662} C_VEL
LIN {X 0,Y 560.92,Z 665.635,A -85,B 0,C 180,E1 -2987.217,E2 -2987.217} C_VEL
LIN {X 0,Y 561.141,Z 651.176,A -85,B 0,C 180,E1 -2987.637,E2 -2987.637} C_VEL
LIN {X 0,Y 561.23,Z 636.688,A -85,B 0,C 180,E1 -2987.922,E2 -2987.922} C_VEL
LIN {X 0,Y 561.804,Z 480.148,A -85,B 0,C 180,E1 -2989.984,E2 -2989.984} C_VEL
LIN {X 0,Y 560.617,Z 473.208,A -85,B 0,C 180,E1 -2990.125,E2 -2990.125} C_VEL
LIN {X 0,Y 561.154,Z 443.059,A -85,B 0,C 180,E1 -2993.04,E2 -2993.04} C_VEL
LIN {X 0,Y 561.538,Z 419.534,A -85,B 0,C 180,E1 -2995.305,E2 -2995.305} C_VEL
LIN {X 0,Y 561.883,Z 388.402,A -85,B 0,C 180,E1 -2998.276,E2 -2998.276} C_VEL
LIN {X 0,Y 561.909,Z 372.611,A -85,B 0,C 180,E1 -2999.812,E2 -2999.812} C_VEL
LIN {X 0,Y 559.149,Z 361.462,A -85,B 0,C 180,E1 -3001.065,E2 -3001.065} C_VEL
LIN {X 0,Y 559.144,Z 361.464,A -85,B 0,C 180,E1 -3003.946,E2 -3003.946} C_VEL
LIN {X 0,Y 559.103,Z 361.461,A -85,B 0,C 180,E1 -3007.11,E2 -3007.11} C_VEL
LIN {X 0,Y 559.147,Z 361.463,A -85,B 0,C 180,E1 -3009.94,E2 -3009.94} C_VEL
LIN {X 0,Y 559.135,Z 361.458,A -85,B 0,C 180,E1 -3012.744,E2 -3012.744} C_VEL
LIN {X 0,Y 559.103,Z 361.461,A -85,B 0,C 180,E1 -3015.764,E2 -3015.764} C_VEL
LIN {X 0,Y 559.088,Z 361.47,A -85,B 0,C 180,E1 -3018.223,E2 -3018.223} C_VEL
LIN {X 0,Y 559.153,Z 361.453,A -85,B 0,C 180,E1 -3021.064,E2 -3021.064} C_VEL
LIN {X 0,Y 559.099,Z 361.464,A -85,B 0,C 180,E1 -3023.786,E2 -3023.786} C_VEL
LIN {X 0,Y 559.122,Z 361.466,A -85,B 0,C 180,E1 -3026.422,E2 -3026.422} C_VEL
LIN {X 0,Y 559.132,Z 361.457,A -85,B 0,C 180,E1 -3028.979,E2 -3028.979} C_VEL
LIN {X 0,Y 559.086,Z 361.464,A -85,B 0,C 180,E1 -3031.631,E2 -3031.631} C_VEL
LIN {X 0,Y 559.139,Z 361.459,A -85,B 0,C 180,E1 -3033.901,E2 -3033.901} C_VEL
LIN {X 0,Y 559.089,Z 361.469,A -85,B 0,C 180,E1 -3036.58,E2 -3036.58} C_VEL
LIN {X 0,Y 559.095,Z 361.46,A -85,B 0,C 180,E1 -3039.392,E2 -3039.392} C_VEL
LIN {X 0,Y 559.092,Z 361.463,A -85,B 0,C 180,E1 -3041.684,E2 -3041.684} C_VEL
LIN {X 0,Y 559.11,Z 361.465,A -85,B 0,C 180,E1 -3044.694,E2 -3044.694} C_VEL
LIN {X 0,Y 559.123,Z 361.458,A -85,B 0,C 180,E1 -3047.662,E2 -3047.662} C_VEL
LIN {X 0,Y 559.097,Z 361.461,A -85,B 0,C 180,E1 -3049.864,E2 -3049.864} C_VEL
LIN {X 0,Y 559.134,Z 361.46,A -85,B 0,C 180,E1 -3052.779,E2 -3052.779} C_VEL
LIN {X 0,Y 559.214,Z 361.45,A -85,B 0,C 180,E1 -3054.953,E2 -3054.953} C_VEL
LIN {X 0,Y 559.215,Z 361.445,A -85,B 0,C 180,E1 -3057.839,E2 -3057.839} C_VEL
LIN {X 0,Y 559.255,Z 361.448,A -85,B 0,C 180,E1 -3060.72,E2 -3060.72} C_VEL
LIN {X 0,Y 559.211,Z 361.452,A -85,B 0,C 180,E1 -3062.882,E2 -3062.882} C_VEL
LIN {X 0,Y 559.187,Z 361.447,A -85,B 0,C 180,E1 -3065.771,E2 -3065.771} C_VEL
LIN {X 0,Y 559.146,Z 361.461,A -85,B 0,C 180,E1 -3068.675,E2 -3068.675} C_VEL
LIN {X 0,Y 559.185,Z 361.449,A -85,B 0,C 180,E1 -3071.601,E2 -3071.601} C_VEL
LIN {X 0,Y 559.166,Z 361.455,A -85,B 0,C 180,E1 -3074.588,E2 -3074.588} C_VEL
LIN {X 0,Y 559.12,Z 361.458,A -85,B 0,C 180,E1 -3077.558,E2 -3077.558} C_VEL
LIN {X 0,Y 559.149,Z 361.452,A -85,B 0,C 180,E1 -3079.838,E2 -3079.838} C_VEL
LIN {X 0,Y 559.12,Z 361.457,A -85,B 0,C 180,E1 -3082.154,E2 -3082.154} C_VEL
LIN {X 0,Y 559.124,Z 361.46,A -85,B 0,C 180,E1 -3085.179,E2 -3085.179} C_VEL
LIN {X 0,Y 559.121,Z 361.46,A -85,B 0,C 180,E1 -3088.375,E2 -3088.375} C_VEL
LIN {X 0,Y 559.116,Z 361.46,A -85,B 0,C 180,E1 -3090.631,E2 -3090.631} C_VEL
LIN {X 0,Y 558.461,Z 361.544,A -85,B 0,C 180,E1 -3091.233,E2 -3091.233} C_VEL
LIN {X 0,Y 555.599,Z 361.901,A -85,B 0,C 180,E1 -3092.209,E2 -3092.209} C_VEL
LIN {X 0,Y 553.181,Z 362.207,A -85,B 0,C 180,E1 -3092.995,E2 -3092.995} C_VEL
LIN {X 0,Y 552.154,Z 362.328,A -85,B 0,C 180,E1 -3093.602,E2 -3093.602} C_VEL
LIN {X 0,Y 552.077,Z 362.336,A -85,B 0,C 180,E1 -3093.807,E2 -3093.807} C_VEL
LIN {X 0,Y 552.095,Z 362.34,A -85,B 0,C 180,E1 -3096.748,E2 -3096.748} C_VEL
LIN {X 0,Y 552.116,Z 362.332,A -85,B 0,C 180,E1 -3099.529,E2 -3099.529} C_VEL
LIN {X 0,Y 552.099,Z 362.335,A -85,B 0,C 180,E1 -3102.429,E2 -3102.429} C_VEL
LIN {X 0,Y 552.084,Z 362.337,A -85,B 0,C 180,E1 -3105.563,E2 -3105.563} C_VEL
LIN {X 0,Y 552.068,Z 362.34,A -85,B 0,C 180,E1 -3108.551,E2 -3108.551} C_VEL
LIN {X 0,Y 552.107,Z 362.335,A -85,B 0,C 180,E1 -3111.412,E2 -3111.412} C_VEL
LIN {X 0,Y 552.066,Z 362.336,A -85,B 0,C 180,E1 -3114.156,E2 -3114.156} C_VEL
LIN {X 0,Y 552.103,Z 362.341,A -85,B 0,C 180,E1 -3117.156,E2 -3117.156} C_VEL
LIN {X 0,Y 552.086,Z 362.337,A -85,B 0,C 180,E1 -3119.956,E2 -3119.956} C_VEL
LIN {X 0,Y 552.078,Z 362.345,A -85,B 0,C 180,E1 -3121.106,E2 -3121.106} C_VEL
LIN {X 0,Y 554.39,Z 368.569,A -85,B 0,C 180,E1 -3121.29,E2 -3121.29} C_VEL
LIN {X 0,Y 554.996,Z 370.052,A -85,B 0,C 180,E1 -3121.334,E2 -3121.334} C_VEL
LIN {X 0,Y 554.457,Z 490.329,A -85,B 0,C 180,E1 -3122.953,E2 -3122.953} C_VEL
LIN {X 0,Y 554.308,Z 505.71,A -85,B 0,C 180,E1 -3123.302,E2 -3123.302} C_VEL
LIN {X 0,Y 554.007,Z 520.617,A -85,B 0,C 180,E1 -3123.789,E2 -3123.789} C_VEL
LIN {X 0,Y 553.726,Z 535.446,A -85,B 0,C 180,E1 -3124.436,E2 -3124.436} C_VEL
LIN {X 0,Y 553.378,Z 549.648,A -85,B 0,C 180,E1 -3125.223,E2 -3125.223} C_VEL
LIN {X 0,Y 553.088,Z 562.593,A -85,B 0,C 180,E1 -3126.107,E2 -3126.107} C_VEL
LIN {X 0,Y 552.722,Z 575.628,A -85,B 0,C 180,E1 -3127.182,E2 -3127.182} C_VEL
LIN {X 0,Y 552.507,Z 587.365,A -85,B 0,C 180,E1 -3128.354,E2 -3128.354} C_VEL
LIN {X 0,Y 552.282,Z 597.141,A -85,B 0,C 180,E1 -3129.517,E2 -3129.517} C_VEL
LIN {X 0,Y 552.039,Z 606.654,A -85,B 0,C 180,E1 -3130.864,E2 -3130.864} C_VEL
LIN {X 0,Y 551.941,Z 614.476,A -85,B 0,C 180,E1 -3132.207,E2 -3132.207} C_VEL
LIN {X 0,Y 551.806,Z 621.705,A -85,B 0,C 180,E1 -3133.729,E2 -3133.729} C_VEL
LIN {X 0,Y 551.767,Z 627.319,A -85,B 0,C 180,E1 -3135.242,E2 -3135.242} C_VEL
LIN {X 0,Y 551.672,Z 631.491,A -85,B 0,C 180,E1 -3136.744,E2 -3136.744} C_VEL
LIN {X 0,Y 551.671,Z 634.359,A -85,B 0,C 180,E1 -3138.24,E2 -3138.24} C_VEL
LIN {X 0,Y 551.671,Z 636.001,A -85,B 0,C 180,E1 -3139.727,E2 -3139.727} C_VEL
LIN {X 0,Y 551.667,Z 636.472,A -85,B 0,C 180,E1 -3141.207,E2 -3141.207} C_VEL
LIN {X 0,Y 551.691,Z 635.786,A -85,B 0,C 180,E1 -3142.682,E2 -3142.682} C_VEL
LIN {X 0,Y 551.744,Z 633.899,A -85,B 0,C 180,E1 -3144.152,E2 -3144.152} C_VEL
LIN {X 0,Y 551.704,Z 630.831,A -85,B 0,C 180,E1 -3145.617,E2 -3145.617} C_VEL
LIN {X 0,Y 551.745,Z 626.533,A -85,B 0,C 180,E1 -3147.08,E2 -3147.08} C_VEL
LIN {X 0,Y 551.761,Z 620.923,A -85,B 0,C 180,E1 -3148.541,E2 -3148.541} C_VEL
LIN {X 0,Y 551.952,Z 613.842,A -85,B 0,C 180,E1 -3150,E2 -3150} C_VEL
LIN {X 0,Y 552.063,Z 606.315,A -85,B 0,C 180,E1 -3151.277,E2 -3151.277} C_VEL
LIN {X 0,Y 552.239,Z 597.308,A -85,B 0,C 180,E1 -3152.553,E2 -3152.553} C_VEL
LIN {X 0,Y 552.522,Z 586.486,A -85,B 0,C 180,E1 -3153.829,E2 -3153.829} C_VEL
LIN {X 0,Y 552.762,Z 575.435,A -85,B 0,C 180,E1 -3154.923,E2 -3154.923} C_VEL
LIN {X 0,Y 553.038,Z 563.365,A -85,B 0,C 180,E1 -3155.927,E2 -3155.927} C_VEL
LIN {X 0,Y 553.386,Z 550.122,A -85,B 0,C 180,E1 -3156.838,E2 -3156.838} C_VEL
LIN {X 0,Y 553.721,Z 536.058,A -85,B 0,C 180,E1 -3157.625,E2 -3157.625} C_VEL
LIN {X 0,Y 554.005,Z 521.936,A -85,B 0,C 180,E1 -3158.251,E2 -3158.251} C_VEL
LIN {X 0,Y 554.253,Z 506.25,A -85,B 0,C 180,E1 -3158.775,E2 -3158.775} C_VEL
LIN {X 0,Y 554.436,Z 490.159,A -85,B 0,C 180,E1 -3159.14,E2 -3159.14} C_VEL
LIN {X 0,Y 554.837,Z 369.565,A -85,B 0,C 180,E1 -3160.768,E2 -3160.768} C_VEL
LIN {X 0,Y 552.138,Z 362.339,A -85,B 0,C 180,E1 -3160.984,E2 -3160.984} C_VEL
LIN {X 0,Y 552.088,Z 362.336,A -85,B 0,C 180,E1 -3163.997,E2 -3163.997} C_VEL
LIN {X 0,Y 552.087,Z 362.342,A -85,B 0,C 180,E1 -3167.025,E2 -3167.025} C_VEL
LIN {X 0,Y 552.093,Z 362.334,A -85,B 0,C 180,E1 -3170.102,E2 -3170.102} C_VEL
LIN {X 0,Y 552.038,Z 362.343,A -85,B 0,C 180,E1 -3172.453,E2 -3172.453} C_VEL
LIN {X 0,Y 552.062,Z 362.344,A -85,B 0,C 180,E1 -3175.329,E2 -3175.329} C_VEL
LIN {X 0,Y 552.047,Z 362.34,A -85,B 0,C 180,E1 -3178.101,E2 -3178.101} C_VEL
LIN {X 0,Y 552.065,Z 362.336,A -85,B 0,C 180,E1 -3180.611,E2 -3180.611} C_VEL
LIN {X 0,Y 552.086,Z 362.342,A -85,B 0,C 180,E1 -3183.187,E2 -3183.187} C_VEL
LIN {X 0,Y 552.061,Z 362.338,A -85,B 0,C 180,E1 -3185.845,E2 -3185.845} C_VEL
LIN {X 0,Y 552.084,Z 362.337,A -85,B 0,C 180,E1 -3188.591,E2 -3188.591} C_VEL
LIN {X 0,Y 552.051,Z 362.344,A -85,B 0,C 180,E1 -3191.451,E2 -3191.451} C_VEL
LIN {X 0,Y 552.062,Z 362.337,A -85,B 0,C 180,E1 -3194.528,E2 -3194.528} C_VEL
LIN {X 0,Y 552.074,Z 362.339,A -85,B 0,C 180,E1 -3197.59,E2 -3197.59} C_VEL
LIN {X 0,Y 552.09,Z 362.334,A -85,B 0,C 180,E1 -3200.469,E2 -3200.469} C_VEL
LIN {X 0,Y 552.088,Z 362.344,A -85,B 0,C 180,E1 -3203.318,E2 -3203.318} C_VEL
LIN {X 0,Y 552.081,Z 362.334,A -85,B 0,C 180,E1 -3205.936,E2 -3205.936} C_VEL
LIN {X 0,Y 552.072,Z 362.337,A -85,B 0,C 180,E1 -3208.537,E2 -3208.537} C_VEL
LIN {X 0,Y 552.067,Z 362.344,A -85,B 0,C 180,E1 -3211.447,E2 -3211.447} C_VEL
LIN {X 0,Y 552.038,Z 362.34,A -85,B 0,C 180,E1 -3214.351,E2 -3214.351} C_VEL
LIN {X 0,Y 552.078,Z 362.335,A -85,B 0,C 180,E1 -3216.757,E2 -3216.757} C_VEL
LIN {X 0,Y 552.104,Z 362.338,A -85,B 0,C 180,E1 -3219.119,E2 -3219.119} C_VEL
LIN {X 0,Y 552.07,Z 362.344,A -85,B 0,C 180,E1 -3221.442,E2 -3221.442} C_VEL
LIN {X 0,Y 552.079,Z 362.34,A -85,B 0,C 180,E1 -3223.736,E2 -3223.736} C_VEL
LIN {X 0,Y 552.101,Z 362.332,A -85,B 0,C 180,E1 -3226.003,E2 -3226.003} C_VEL
LIN {X 0,Y 552.14,Z 362.323,A -85,B 0,C 180,E1 -3228.993,E2 -3228.993} C_VEL
LIN {X 0,Y 552.093,Z 362.334,A -85,B 0,C 180,E1 -3231.95,E2 -3231.95} C_VEL
LIN {X 0,Y 552.202,Z 362.321,A -85,B 0,C 180,E1 -3234.889,E2 -3234.889} C_VEL
LIN {X 0,Y 552.194,Z 362.324,A -85,B 0,C 180,E1 -3237.812,E2 -3237.812} C_VEL
LIN {X 0,Y 552.196,Z 362.323,A -85,B 0,C 180,E1 -3240,E2 -3240} C_VEL
LIN {X 0,Y 552.171,Z 362.324,A -85,B 0,C 180,E1 -3242.918,E2 -3242.918} C_VEL
LIN {X 0,Y 552.158,Z 362.331,A -85,B 0,C 180,E1 -3245.844,E2 -3245.844} C_VEL
LIN {X 0,Y 552.106,Z 362.33,A -85,B 0,C 180,E1 -3248.786,E2 -3248.786} C_VEL
LIN {X 0,Y 552.137,Z 362.336,A -85,B 0,C 180,E1 -3251.751,E2 -3251.751} C_VEL
LIN {X 0,Y 552.108,Z 362.33,A -85,B 0,C 180,E1 -3254.749,E2 -3254.749} C_VEL
LIN {X 0,Y 552.063,Z 362.344,A -85,B 0,C 180,E1 -3257.79,E2 -3257.79} C_VEL
LIN {X 0,Y 552.081,Z 362.339,A -85,B 0,C 180,E1 -3260.103,E2 -3260.103} C_VEL
LIN {X 0,Y 552.032,Z 362.34,A -85,B 0,C 180,E1 -3262.453,E2 -3262.453} C_VEL
LIN {X 0,Y 552.073,Z 362.34,A -85,B 0,C 180,E1 -3265.334,E2 -3265.334} C_VEL
LIN {X 0,Y 552.038,Z 362.344,A -85,B 0,C 180,E1 -3268.102,E2 -3268.102} C_VEL
LIN {X 0,Y 552.079,Z 362.336,A -85,B 0,C 180,E1 -3270.611,E2 -3270.611} C_VEL
LIN {X 0,Y 552.085,Z 362.335,A -85,B 0,C 180,E1 -3273.188,E2 -3273.188} C_VEL
LIN {X 0,Y 552.058,Z 362.348,A -85,B 0,C 180,E1 -3275.846,E2 -3275.846} C_VEL
LIN {X 0,Y 552.079,Z 362.334,A -85,B 0,C 180,E1 -3278.592,E2 -3278.592} C_VEL
LIN {X 0,Y 552.052,Z 362.343,A -85,B 0,C 180,E1 -3281.452,E2 -3281.452} C_VEL
LIN {X 0,Y 552.06,Z 362.339,A -85,B 0,C 180,E1 -3284.529,E2 -3284.529} C_VEL
LIN {X 0,Y 552.079,Z 362.341,A -85,B 0,C 180,E1 -3287.59,E2 -3287.59} C_VEL
LIN {X 0,Y 552.106,Z 362.332,A -85,B 0,C 180,E1 -3290.941,E2 -3290.941} C_VEL
LIN {X 0,Y 552.045,Z 362.342,A -85,B 0,C 180,E1 -3293.326,E2 -3293.326} C_VEL
LIN {X 0,Y 552.091,Z 362.343,A -85,B 0,C 180,E1 -3295.937,E2 -3295.937} C_VEL
LIN {X 0,Y 552.112,Z 362.518,A -85,B 0,C 180,E1 -3298.696,E2 -3298.696} C_VEL
LIN {X 0,Y 555.145,Z 374.081,A -85,B 0,C 180,E1 -3300.009,E2 -3300.009} C_VEL
LIN {X 0,Y 555.021,Z 394.895,A -85,B 0,C 180,E1 -3302.063,E2 -3302.063} C_VEL
LIN {X 0,Y 554.602,Z 425.056,A -85,B 0,C 180,E1 -3304.981,E2 -3304.981} C_VEL
LIN {X 0,Y 554.192,Z 454.404,A -85,B 0,C 180,E1 -3307.782,E2 -3307.782} C_VEL
LIN {X 0,Y 553.793,Z 473.204,A -85,B 0,C 180,E1 -3309.615,E2 -3309.615} C_VEL
LIN {X 0,Y 555.182,Z 482.686,A -85,B 0,C 180,E1 -3309.802,E2 -3309.802} C_VEL
LIN {X 0,Y 554.47,Z 641.094,A -85,B 0,C 180,E1 -3311.922,E2 -3311.922} C_VEL
LIN {X 0,Y 554.28,Z 656.709,A -85,B 0,C 180,E1 -3312.284,E2 -3312.284} C_VEL
LIN {X 0,Y 554.04,Z 672.04,A -85,B 0,C 180,E1 -3312.8,E2 -3312.8} C_VEL
LIN {X 0,Y 553.795,Z 685.78,A -85,B 0,C 180,E1 -3313.409,E2 -3313.409} C_VEL
LIN {X 0,Y 553.405,Z 699.252,A -85,B 0,C 180,E1 -3314.155,E2 -3314.155} C_VEL
LIN {X 0,Y 553.086,Z 712.287,A -85,B 0,C 180,E1 -3315.04,E2 -3315.04} C_VEL
LIN {X 0,Y 552.78,Z 724.294,A -85,B 0,C 180,E1 -3316.021,E2 -3316.021} C_VEL
LIN {X 0,Y 552.529,Z 735.75,A -85,B 0,C 180,E1 -3317.139,E2 -3317.139} C_VEL
LIN {X 0,Y 552.252,Z 746.437,A -85,B 0,C 180,E1 -3318.383,E2 -3318.383} C_VEL
LIN {X 0,Y 552.124,Z 754.855,A -85,B 0,C 180,E1 -3319.549,E2 -3319.549} C_VEL
LIN {X 0,Y 551.959,Z 762.735,A -85,B 0,C 180,E1 -3320.842,E2 -3320.842} C_VEL
LIN {X 0,Y 551.837,Z 770.09,A -85,B 0,C 180,E1 -3322.315,E2 -3322.315} C_VEL
LIN {X 0,Y 551.758,Z 775.607,A -85,B 0,C 180,E1 -3323.691,E2 -3323.691} C_VEL
LIN {X 0,Y 551.713,Z 779.386,A -85,B 0,C 180,E1 -3324.884,E2 -3324.884} C_VEL
LIN {X 0,Y 551.73,Z 782.888,A -85,B 0,C 180,E1 -3326.348,E2 -3326.348} C_VEL
LIN {X 0,Y 551.653,Z 785.191,A -85,B 0,C 180,E1 -3327.809,E2 -3327.809} C_VEL
LIN {X 0,Y 551.639,Z 786.348,A -85,B 0,C 180,E1 -3329.27,E2 -3329.27} C_VEL
LIN {X 0,Y 551.639,Z 786.348,A -85,B 0,C 180,E1 -3330.73,E2 -3330.73} C_VEL
LIN {X 0,Y 551.653,Z 785.189,A -85,B 0,C 180,E1 -3332.19,E2 -3332.19} C_VEL
LIN {X 0,Y 551.73,Z 782.886,A -85,B 0,C 180,E1 -3333.651,E2 -3333.651} C_VEL
LIN {X 0,Y 551.713,Z 779.387,A -85,B 0,C 180,E1 -3335.115,E2 -3335.115} C_VEL
LIN {X 0,Y 551.779,Z 774.611,A -85,B 0,C 180,E1 -3336.582,E2 -3336.582} C_VEL
LIN {X 0,Y 551.876,Z 768.424,A -85,B 0,C 180,E1 -3338.052,E2 -3338.052} C_VEL
LIN {X 0,Y 551.951,Z 760.649,A -85,B 0,C 180,E1 -3339.527,E2 -3339.527} C_VEL
LIN {X 0,Y 552.183,Z 752.372,A -85,B 0,C 180,E1 -3340.82,E2 -3340.82} C_VEL
LIN {X 0,Y 552.351,Z 742.396,A -85,B 0,C 180,E1 -3342.118,E2 -3342.118} C_VEL
LIN {X 0,Y 552.608,Z 732.193,A -85,B 0,C 180,E1 -3343.233,E2 -3343.233} C_VEL
LIN {X 0,Y 552.906,Z 720.027,A -85,B 0,C 180,E1 -3344.351,E2 -3344.351} C_VEL
LIN {X 0,Y 553.243,Z 707.453,A -85,B 0,C 180,E1 -3345.309,E2 -3345.309} C_VEL
LIN {X 0,Y 553.514,Z 694.521,A -85,B 0,C 180,E1 -3346.125,E2 -3346.125} C_VEL
LIN {X 0,Y 553.86,Z 679.841,A -85,B 0,C 180,E1 -3346.873,E2 -3346.873} C_VEL
LIN {X 0,Y 554.134,Z 665.635,A -85,B 0,C 180,E1 -3347.435,E2 -3347.435} C_VEL
LIN {X 0,Y 554.397,Z 650.537,A -85,B 0,C 180,E1 -3347.875,E2 -3347.875} C_VEL
LIN {X 0,Y 554.5,Z 636.352,A -85,B 0,C 180,E1 -3348.153,E2 -3348.153} C_VEL
LIN {X 0,Y 555.19,Z 481.886,A -85,B 0,C 180,E1 -3350.209,E2 -3350.209} C_VEL
LIN {X 0,Y 553.804,Z 473.213,A -85,B 0,C 180,E1 -3350.383,E2 -3350.383} C_VEL
LIN {X 0,Y 554.318,Z 444.832,A -85,B 0,C 180,E1 -3353.143,E2 -3353.143} C_VEL
LIN {X 0,Y 554.743,Z 414.218,A -85,B 0,C 180,E1 -3356.052,E2 -3356.052} C_VEL
LIN {X 0,Y 555.022,Z 387.393,A -85,B 0,C 180,E1 -3358.658,E2 -3358.658} C_VEL
LIN {X 0,Y 555.103,Z 373.927,A -85,B 0,C 180,E1 -3359.988,E2 -3359.988} C_VEL
LIN {X 0,Y 552.116,Z 362.34,A -85,B 0,C 180,E1 -3361.325,E2 -3361.325} C_VEL
LIN {X 0,Y 552.087,Z 362.343,A -85,B 0,C 180,E1 -3364.163,E2 -3364.163} C_VEL
LIN {X 0,Y 552.043,Z 362.342,A -85,B 0,C 180,E1 -3366.75,E2 -3366.75} C_VEL
LIN {X 0,Y 552.116,Z 362.334,A -85,B 0,C 180,E1 -3369.527,E2 -3369.527} C_VEL
LIN {X 0,Y 552.098,Z 362.338,A -85,B 0,C 180,E1 -3372.427,E2 -3372.427} C_VEL
LIN {X 0,Y 552.055,Z 362.336,A -85,B 0,C 180,E1 -3375.558,E2 -3375.558} C_VEL
LIN {X 0,Y 552.048,Z 362.343,A -85,B 0,C 180,E1 -3378.548,E2 -3378.548} C_VEL
LIN {X 0,Y 552.096,Z 362.332,A -85,B 0,C 180,E1 -3381.409,E2 -3381.409} C_VEL
LIN {X 0,Y 552.049,Z 362.344,A -85,B 0,C 180,E1 -3384.562,E2 -3384.562} C_VEL
LIN {X 0,Y 552.082,Z 362.335,A -85,B 0,C 180,E1 -3387.156,E2 -3387.156} C_VEL
LIN {X 0,Y 552.073,Z 362.34,A -85,B 0,C 180,E1 -3389.954,E2 -3389.954} C_VEL
LIN {X 0,Y 552.062,Z 362.339,A -85,B 0,C 180,E1 -3393.012,E2 -3393.012} C_VEL
LIN {X 0,Y 552.059,Z 362.341,A -85,B 0,C 180,E1 -3395.96,E2 -3395.96} C_VEL
LIN {X 0,Y 552.054,Z 362.338,A -85,B 0,C 180,E1 -3399.117,E2 -3399.117} C_VEL
LIN {X 0,Y 552.051,Z 362.339,A -85,B 0,C 180,E1 -3401.442,E2 -3401.442} C_VEL
LIN {X 0,Y 552.055,Z 362.339,A -85,B 0,C 180,E1 -3403.736,E2 -3403.736} C_VEL
LIN {X 0,Y 552.081,Z 362.338,A -85,B 0,C 180,E1 -3406.003,E2 -3406.003} C_VEL
LIN {X 0,Y 552.134,Z 362.33,A -85,B 0,C 180,E1 -3408.993,E2 -3408.993} C_VEL
LIN {X 0,Y 552.115,Z 362.333,A -85,B 0,C 180,E1 -3411.951,E2 -3411.951} C_VEL
LIN {X 0,Y 552.19,Z 362.326,A -85,B 0,C 180,E1 -3414.889,E2 -3414.889} C_VEL
LIN {X 0,Y 552.189,Z 362.32,A -85,B 0,C 180,E1 -3417.812,E2 -3417.812} C_VEL
LIN {X 0,Y 552.225,Z 362.323,A -85,B 0,C 180,E1 -3420.729,E2 -3420.729} C_VEL
LIN {X 0,Y 552.176,Z 362.328,A -85,B 0,C 180,E1 -3422.918,E2 -3422.918} C_VEL
LIN {X 0,Y 552.16,Z 362.322,A -85,B 0,C 180,E1 -3425.845,E2 -3425.845} C_VEL
LIN {X 0,Y 552.118,Z 362.338,A -85,B 0,C 180,E1 -3428.787,E2 -3428.787} C_VEL
LIN {X 0,Y 552.142,Z 362.327,A -85,B 0,C 180,E1 -3431.751,E2 -3431.751} C_VEL
LIN {X 0,Y 552.114,Z 362.334,A -85,B 0,C 180,E1 -3434.749,E2 -3434.749} C_VEL
LIN {X 0,Y 552.078,Z 362.335,A -85,B 0,C 180,E1 -3437.79,E2 -3437.79} C_VEL
LIN {X 0,Y 552.111,Z 362.33,A -85,B 0,C 180,E1 -3440.102,E2 -3440.102} C_VEL
LIN {X 0,Y 552.072,Z 362.338,A -85,B 0,C 180,E1 -3442.452,E2 -3442.452} C_VEL
LIN {X 0,Y 552.067,Z 362.337,A -85,B 0,C 180,E1 -3445.334,E2 -3445.334} C_VEL
LIN {X 0,Y 552.063,Z 362.336,A -85,B 0,C 180,E1 -3448.101,E2 -3448.101} C_VEL
LIN {X 0,Y 552.08,Z 362.341,A -85,B 0,C 180,E1 -3450.629,E2 -3450.629} C_VEL
LIN {X 0,Y 552.093,Z 362.339,A -85,B 0,C 180,E1 -3453.188,E2 -3453.188} C_VEL
LIN {X 0,Y 552.077,Z 362.336,A -85,B 0,C 180,E1 -3453.807,E2 -3453.807} C_VEL
LIN {X 0,Y 551.439,Z 362.42,A -85,B 0,C 180,E1 -3454.416,E2 -3454.416} C_VEL
LIN {X 0,Y 548.625,Z 362.772,A -85,B 0,C 180,E1 -3455.404,E2 -3455.404} C_VEL
LIN {X 0,Y 546.214,Z 363.074,A -85,B 0,C 180,E1 -3456.199,E2 -3456.199} C_VEL
LIN {X 0,Y 545.15,Z 363.205,A -85,B 0,C 180,E1 -3456.813,E2 -3456.813} C_VEL
LIN {X 0,Y 545.048,Z 363.217,A -85,B 0,C 180,E1 -3457.021,E2 -3457.021} C_VEL
LIN {X 0,Y 545.053,Z 363.21,A -85,B 0,C 180,E1 -3460.144,E2 -3460.144} C_VEL
LIN {X 0,Y 545.014,Z 363.22,A -85,B 0,C 180,E1 -3463.113,E2 -3463.113} C_VEL
LIN {X 0,Y 545.042,Z 363.213,A -85,B 0,C 180,E1 -3466.227,E2 -3466.227} C_VEL
LIN {X 0,Y 545.022,Z 363.223,A -85,B 0,C 180,E1 -3468.882,E2 -3468.882} C_VEL
LIN {X 0,Y 545.041,Z 363.212,A -85,B 0,C 180,E1 -3471.763,E2 -3471.763} C_VEL
LIN {X 0,Y 545.021,Z 363.216,A -85,B 0,C 180,E1 -3474.532,E2 -3474.532} C_VEL
LIN {X 0,Y 545.058,Z 363.218,A -85,B 0,C 180,E1 -3477.212,E2 -3477.212} C_VEL
LIN {X 0,Y 545.059,Z 363.214,A -85,B 0,C 180,E1 -3479.811,E2 -3479.811} C_VEL
LIN {X 0,Y 545.044,Z 363.219,A -85,B 0,C 180,E1 -3480.827,E2 -3480.827} C_VEL
LIN {X 0,Y 546.779,Z 367.957,A -85,B 0,C 180,E1 -3480.979,E2 -3480.979} C_VEL
LIN {X 0,Y 548.316,Z 371.651,A -85,B 0,C 180,E1 -3481.092,E2 -3481.092} C_VEL
LIN {X 0,Y 547.772,Z 492.11,A -85,B 0,C 180,E1 -3482.738,E2 -3482.738} C_VEL
LIN {X 0,Y 547.603,Z 507.585,A -85,B 0,C 180,E1 -3483.103,E2 -3483.103} C_VEL
LIN {X 0,Y 547.277,Z 522.238,A -85,B 0,C 180,E1 -3483.601,E2 -3483.601} C_VEL
LIN {X 0,Y 546.937,Z 536.543,A -85,B 0,C 180,E1 -3484.248,E2 -3484.248} C_VEL
LIN {X 0,Y 546.525,Z 551.172,A -85,B 0,C 180,E1 -3485.094,E2 -3485.094} C_VEL
LIN {X 0,Y 546.148,Z 564.018,A -85,B 0,C 180,E1 -3486.015,E2 -3486.015} C_VEL
LIN {X 0,Y 545.746,Z 577.425,A -85,B 0,C 180,E1 -3487.174,E2 -3487.174} C_VEL
LIN {X 0,Y 545.472,Z 588.416,A -85,B 0,C 180,E1 -3488.309,E2 -3488.309} C_VEL
LIN {X 0,Y 545.253,Z 597.702,A -85,B 0,C 180,E1 -3489.438,E2 -3489.438} C_VEL
LIN {X 0,Y 544.976,Z 607.112,A -85,B 0,C 180,E1 -3490.802,E2 -3490.802} C_VEL
LIN {X 0,Y 544.879,Z 614.963,A -85,B 0,C 180,E1 -3492.182,E2 -3492.182} C_VEL
LIN {X 0,Y 544.731,Z 621.177,A -85,B 0,C 180,E1 -3493.511,E2 -3493.511} C_VEL
LIN {X 0,Y 544.688,Z 626.917,A -85,B 0,C 180,E1 -3495.046,E2 -3495.046} C_VEL
LIN {X 0,Y 544.604,Z 631.204,A -85,B 0,C 180,E1 -3496.569,E2 -3496.569} C_VEL
LIN {X 0,Y 544.566,Z 634.177,A -85,B 0,C 180,E1 -3498.084,E2 -3498.084} C_VEL
LIN {X 0,Y 544.575,Z 635.924,A -85,B 0,C 180,E1 -3499.591,E2 -3499.591} C_VEL
LIN {X 0,Y 544.559,Z 636.496,A -85,B 0,C 180,E1 -3501.091,E2 -3501.091} C_VEL
LIN {X 0,Y 544.603,Z 635.869,A -85,B 0,C 180,E1 -3502.586,E2 -3502.586} C_VEL
LIN {X 0,Y 544.642,Z 634.076,A -85,B 0,C 180,E1 -3504.075,E2 -3504.075} C_VEL
LIN {X 0,Y 544.602,Z 631.113,A -85,B 0,C 180,E1 -3505.56,E2 -3505.56} C_VEL
LIN {X 0,Y 544.673,Z 626.922,A -85,B 0,C 180,E1 -3507.042,E2 -3507.042} C_VEL
LIN {X 0,Y 544.673,Z 621.428,A -85,B 0,C 180,E1 -3508.522,E2 -3508.522} C_VEL
LIN {X 0,Y 544.871,Z 614.474,A -85,B 0,C 180,E1 -3510,E2 -3510} C_VEL
LIN {X 0,Y 545.013,Z 607.078,A -85,B 0,C 180,E1 -3511.293,E2 -3511.293} C_VEL
LIN {X 0,Y 545.21,Z 598.194,A -85,B 0,C 180,E1 -3512.586,E2 -3512.586} C_VEL
LIN {X 0,Y 545.528,Z 587.567,A -85,B 0,C 180,E1 -3513.878,E2 -3513.878} C_VEL
LIN {X 0,Y 545.806,Z 575.712,A -85,B 0,C 180,E1 -3515.079,E2 -3515.079} C_VEL
LIN {X 0,Y 546.187,Z 562.546,A -85,B 0,C 180,E1 -3516.187,E2 -3516.187} C_VEL
LIN {X 0,Y 546.602,Z 549.343,A -85,B 0,C 180,E1 -3517.109,E2 -3517.109} C_VEL
LIN {X 0,Y 546.949,Z 535.777,A -85,B 0,C 180,E1 -3517.878,E2 -3517.878} C_VEL
LIN {X 0,Y 547.31,Z 521.095,A -85,B 0,C 180,E1 -3518.529,E2 -3518.529} C_VEL
LIN {X 0,Y 547.56,Z 506.258,A -85,B 0,C 180,E1 -3519.023,E2 -3519.023} C_VEL
LIN {X 0,Y 547.73,Z 491.115,A -85,B 0,C 180,E1 -3519.369,E2 -3519.369} C_VEL
LIN {X 0,Y 548.261,Z 371.462,A -85,B 0,C 180,E1 -3521.002,E2 -3521.002} C_VEL
LIN {X 0,Y 545.249,Z 363.991,A -85,B 0,C 180,E1 -3521.226,E2 -3521.226} C_VEL
LIN {X 0,Y 545.112,Z 363.212,A -85,B 0,C 180,E1 -3521.257,E2 -3521.257} C_VEL
LIN {X 0,Y 545.061,Z 363.217,A -85,B 0,C 180,E1 -3524.748,E2 -3524.748} C_VEL
LIN {X 0,Y 545.045,Z 363.212,A -85,B 0,C 180,E1 -3528.027,E2 -3528.027} C_VEL
LIN {X 0,Y 545.03,Z 363.215,A -85,B 0,C 180,E1 -3530.374,E2 -3530.374} C_VEL
LIN {X 0,Y 544.984,Z 363.225,A -85,B 0,C 180,E1 -3532.76,E2 -3532.76} C_VEL
LIN {X 0,Y 545.014,Z 363.219,A -85,B 0,C 180,E1 -3535.49,E2 -3535.49} C_VEL
LIN {X 0,Y 544.997,Z 363.22,A -85,B 0,C 180,E1 -3537.66,E2 -3537.66} C_VEL
LIN {X 0,Y 545.019,Z 363.211,A -85,B 0,C 180,E1 -3540.235,E2 -3540.235} C_VEL
LIN {X 0,Y 545.056,Z 363.22,A -85,B 0,C 180,E1 -3543.058,E2 -3543.058} C_VEL
LIN {X 0,Y 545.012,Z 363.218,A -85,B 0,C 180,E1 -3545.669,E2 -3545.669} C_VEL
LIN {X 0,Y 545.027,Z 363.214,A -85,B 0,C 180,E1 -3548.239,E2 -3548.239} C_VEL
LIN {X 0,Y 545.001,Z 363.225,A -85,B 0,C 180,E1 -3551.121,E2 -3551.121} C_VEL
LIN {X 0,Y 545.02,Z 363.213,A -85,B 0,C 180,E1 -3554.132,E2 -3554.132} C_VEL
LIN {X 0,Y 545.011,Z 363.22,A -85,B 0,C 180,E1 -3556.886,E2 -3556.886} C_VEL
LIN {X 0,Y 545.046,Z 363.213,A -85,B 0,C 180,E1 -3559.855,E2 -3559.855} C_VEL
LIN {X 0,Y 545.027,Z 363.22,A -85,B 0,C 180,E1 -3563.079,E2 -3563.079} C_VEL
LIN {X 0,Y 545.042,Z 363.214,A -85,B 0,C 180,E1 -3565.611,E2 -3565.611} C_VEL
LIN {X 0,Y 545.035,Z 363.213,A -85,B 0,C 180,E1 -3568.323,E2 -3568.323} C_VEL
LIN {X 0,Y 545.028,Z 363.22,A -85,B 0,C 180,E1 -3571.503,E2 -3571.503} C_VEL
LIN {X 0,Y 545.007,Z 363.217,A -85,B 0,C 180,E1 -3573.995,E2 -3573.995} C_VEL
LIN {X 0,Y 545.06,Z 363.208,A -85,B 0,C 180,E1 -3576.439,E2 -3576.439} C_VEL
LIN {X 0,Y 545.079,Z 363.212,A -85,B 0,C 180,E1 -3579.627,E2 -3579.627} C_VEL
LIN {X 0,Y 545.04,Z 363.212,A -85,B 0,C 180,E1 -3582.748,E2 -3582.748} C_VEL
LIN {X 0,Y 545.059,Z 363.211,A -85,B 0,C 180,E1 -3585.819,E2 -3585.819} C_VEL
LIN {X 0,Y 545.098,Z 363.198,A -85,B 0,C 180,E1 -3588.849,E2 -3588.849} C_VEL
LIN {X 0,Y 545.051,Z 363.213,A -85,B 0,C 180,E1 -3591.846,E2 -3591.846} C_VEL
LIN {X 0,Y 545.158,Z 363.198,A -85,B 0,C 180,E1 -3594.822,E2 -3594.822} C_VEL
LIN {X 0,Y 545.168,Z 363.199,A -85,B 0,C 180,E1 -3597.783,E2 -3597.783} C_VEL
LIN {X 0,Y 545.166,Z 363.199,A -85,B 0,C 180,E1 -3600,E2 -3600} C_VEL
LIN {X 0,Y 545.14,Z 363.2,A -85,B 0,C 180,E1 -3602.956,E2 -3602.956} C_VEL
LIN {X 0,Y 545.106,Z 363.208,A -85,B 0,C 180,E1 -3605.92,E2 -3605.92} C_VEL
LIN {X 0,Y 545.05,Z 363.21,A -85,B 0,C 180,E1 -3608.901,E2 -3608.901} C_VEL
LIN {X 0,Y 545.079,Z 363.212,A -85,B 0,C 180,E1 -3611.905,E2 -3611.905} C_VEL
LIN {X 0,Y 545.064,Z 363.208,A -85,B 0,C 180,E1 -3614.944,E2 -3614.944} C_VEL
LIN {X 0,Y 545.031,Z 363.216,A -85,B 0,C 180,E1 -3618.027,E2 -3618.027} C_VEL
LIN {X 0,Y 545.018,Z 363.216,A -85,B 0,C 180,E1 -3620.375,E2 -3620.375} C_VEL
LIN {X 0,Y 544.98,Z 363.218,A -85,B 0,C 180,E1 -3622.76,E2 -3622.76} C_VEL
LIN {X 0,Y 545.025,Z 363.22,A -85,B 0,C 180,E1 -3625.496,E2 -3625.496} C_VEL
LIN {X 0,Y 545.022,Z 363.215,A -85,B 0,C 180,E1 -3628.497,E2 -3628.497} C_VEL
LIN {X 0,Y 545.043,Z 363.213,A -85,B 0,C 180,E1 -3631.049,E2 -3631.049} C_VEL
LIN {X 0,Y 545.032,Z 363.219,A -85,B 0,C 180,E1 -3633.674,E2 -3633.674} C_VEL
LIN {X 0,Y 544.994,Z 363.22,A -85,B 0,C 180,E1 -3636.384,E2 -3636.384} C_VEL
LIN {X 0,Y 545.036,Z 363.213,A -85,B 0,C 180,E1 -3639.316,E2 -3639.316} C_VEL
LIN {X 0,Y 545.023,Z 363.219,A -85,B 0,C 180,E1 -3642.108,E2 -3642.108} C_VEL
LIN {X 0,Y 545.01,Z 363.217,A -85,B 0,C 180,E1 -3645.172,E2 -3645.172} C_VEL
LIN {X 0,Y 545.027,Z 363.22,A -85,B 0,C 180,E1 -3647.893,E2 -3647.893} C_VEL
LIN {X 0,Y 545.056,Z 363.211,A -85,B 0,C 180,E1 -3650.817,E2 -3650.817} C_VEL
LIN {X 0,Y 544.997,Z 363.224,A -85,B 0,C 180,E1 -3653.617,E2 -3653.617} C_VEL
LIN {X 0,Y 545.038,Z 363.22,A -85,B 0,C 180,E1 -3656.327,E2 -3656.327} C_VEL
LIN {X 0,Y 545.074,Z 363.346,A -85,B 0,C 180,E1 -3658.433,E2 -3658.433} C_VEL
LIN {X 0,Y 548.316,Z 375.711,A -85,B 0,C 180,E1 -3659.858,E2 -3659.858} C_VEL
LIN {X 0,Y 548.315,Z 386.606,A -85,B 0,C 180,E1 -3660.958,E2 -3660.958} C_VEL
LIN {X 0,Y 547.912,Z 414.068,A -85,B 0,C 180,E1 -3663.671,E2 -3663.671} C_VEL
LIN {X 0,Y 547.407,Z 442.797,A -85,B 0,C 180,E1 -3666.447,E2 -3666.447} C_VEL
LIN {X 0,Y 547.024,Z 468.707,A -85,B 0,C 180,E1 -3668.916,E2 -3668.916} C_VEL
LIN {X 0,Y 547.028,Z 473.543,A -85,B 0,C 180,E1 -3669.362,E2 -3669.362} C_VEL
LIN {X 0,Y 548.528,Z 483.917,A -85,B 0,C 180,E1 -3669.563,E2 -3669.563} C_VEL
LIN {X 0,Y 547.735,Z 641.516,A -85,B 0,C 180,E1 -3671.7,E2 -3671.7} C_VEL
LIN {X 0,Y 547.504,Z 656.708,A -85,B 0,C 180,E1 -3672.057,E2 -3672.057} C_VEL
LIN {X 0,Y 547.256,Z 672.038,A -85,B 0,C 180,E1 -3672.58,E2 -3672.58} C_VEL
LIN {X 0,Y 546.96,Z 685.782,A -85,B 0,C 180,E1 -3673.196,E2 -3673.196} C_VEL
LIN {X 0,Y 546.528,Z 699.254,A -85,B 0,C 180,E1 -3673.95,E2 -3673.95} C_VEL
LIN {X 0,Y 546.151,Z 713.128,A -85,B 0,C 180,E1 -3674.908,E2 -3674.908} C_VEL
LIN {X 0,Y 545.818,Z 725.354,A -85,B 0,C 180,E1 -3675.934,E2 -3675.934} C_VEL
LIN {X 0,Y 545.511,Z 737.509,A -85,B 0,C 180,E1 -3677.16,E2 -3677.16} C_VEL
LIN {X 0,Y 545.175,Z 748.103,A -85,B 0,C 180,E1 -3678.446,E2 -3678.446} C_VEL
LIN {X 0,Y 545.05,Z 757.295,A -85,B 0,C 180,E1 -3679.788,E2 -3679.788} C_VEL
LIN {X 0,Y 544.845,Z 764.75,A -85,B 0,C 180,E1 -3681.095,E2 -3681.095} C_VEL
LIN {X 0,Y 544.745,Z 771.7,A -85,B 0,C 180,E1 -3682.587,E2 -3682.587} C_VEL
LIN {X 0,Y 544.706,Z 777.162,A -85,B 0,C 180,E1 -3684.075,E2 -3684.075} C_VEL
LIN {X 0,Y 544.606,Z 781.291,A -85,B 0,C 180,E1 -3685.559,E2 -3685.559} C_VEL
LIN {X 0,Y 544.644,Z 784.185,A -85,B 0,C 180,E1 -3687.041,E2 -3687.041} C_VEL
LIN {X 0,Y 544.543,Z 785.91,A -85,B 0,C 180,E1 -3688.521,E2 -3688.521} C_VEL
LIN {X 0,Y 544.538,Z 786.5,A -85,B 0,C 180,E1 -3690,E2 -3690} C_VEL
LIN {X 0,Y 544.543,Z 785.909,A -85,B 0,C 180,E1 -3691.479,E2 -3691.479} C_VEL
LIN {X 0,Y 544.644,Z 784.183,A -85,B 0,C 180,E1 -3692.958,E2 -3692.958} C_VEL
LIN {X 0,Y 544.606,Z 781.29,A -85,B 0,C 180,E1 -3694.44,E2 -3694.44} C_VEL
LIN {X 0,Y 544.701,Z 777.166,A -85,B 0,C 180,E1 -3695.924,E2 -3695.924} C_VEL
LIN {X 0,Y 544.745,Z 771.703,A -85,B 0,C 180,E1 -3697.412,E2 -3697.412} C_VEL
LIN {X 0,Y 544.845,Z 764.748,A -85,B 0,C 180,E1 -3698.904,E2 -3698.904} C_VEL
LIN {X 0,Y 545.073,Z 756.087,A -85,B 0,C 180,E1 -3700.399,E2 -3700.399} C_VEL
LIN {X 0,Y 545.235,Z 746.711,A -85,B 0,C 180,E1 -3701.734,E2 -3701.734} C_VEL
LIN {X 0,Y 545.51,Z 737.513,A -85,B 0,C 180,E1 -3702.84,E2 -3702.84} C_VEL
LIN {X 0,Y 545.827,Z 725.365,A -85,B 0,C 180,E1 -3704.065,E2 -3704.065} C_VEL
LIN {X 0,Y 546.191,Z 712.814,A -85,B 0,C 180,E1 -3705.115,E2 -3705.115} C_VEL
LIN {X 0,Y 546.558,Z 699.262,A -85,B 0,C 180,E1 -3706.048,E2 -3706.048} C_VEL
LIN {X 0,Y 546.916,Z 685.787,A -85,B 0,C 180,E1 -3706.805,E2 -3706.805} C_VEL
LIN {X 0,Y 547.222,Z 672.062,A -85,B 0,C 180,E1 -3707.421,E2 -3707.421} C_VEL
LIN {X 0,Y 547.513,Z 656.743,A -85,B 0,C 180,E1 -3707.942,E2 -3707.942} C_VEL
LIN {X 0,Y 547.719,Z 641.12,A -85,B 0,C 180,E1 -3708.308,E2 -3708.308} C_VEL
LIN {X 0,Y 548.559,Z 482.73,A -85,B 0,C 180,E1 -3710.452,E2 -3710.452} C_VEL
LIN {X 0,Y 547,Z 473.124,A -85,B 0,C 180,E1 -3710.656,E2 -3710.656} C_VEL
LIN {X 0,Y 547.411,Z 442.716,A -85,B 0,C 180,E1 -3713.552,E2 -3713.552} C_VEL
LIN {X 0,Y 547.925,Z 413.936,A -85,B 0,C 180,E1 -3716.329,E2 -3716.329} C_VEL
LIN {X 0,Y 548.366,Z 383.142,A -85,B 0,C 180,E1 -3719.366,E2 -3719.366} C_VEL
LIN {X 0,Y 548.25,Z 375.472,A -85,B 0,C 180,E1 -3720.144,E2 -3720.144} C_VEL
LIN {X 0,Y 545.068,Z 363.219,A -85,B 0,C 180,E1 -3721.571,E2 -3721.571} C_VEL
LIN {X 0,Y 545.037,Z 363.217,A -85,B 0,C 180,E1 -3724.565,E2 -3724.565} C_VEL
LIN {X 0,Y 545.003,Z 363.218,A -85,B 0,C 180,E1 -3727.305,E2 -3727.305} C_VEL
LIN {X 0,Y 545.048,Z 363.221,A -85,B 0,C 180,E1 -3730.143,E2 -3730.143} C_VEL
LIN {X 0,Y 545.013,Z 363.215,A -85,B 0,C 180,E1 -3733.111,E2 -3733.111} C_VEL
LIN {X 0,Y 545.012,Z 363.22,A -85,B 0,C 180,E1 -3736.228,E2 -3736.228} C_VEL
LIN {X 0,Y 545.003,Z 363.217,A -85,B 0,C 180,E1 -3738.878,E2 -3738.878} C_VEL
LIN {X 0,Y 545.061,Z 363.21,A -85,B 0,C 180,E1 -3740.817,E2 -3740.817} C_VEL
LIN {X 0,Y 544.989,Z 363.22,A -85,B 0,C 180,E1 -3743.616,E2 -3743.616} C_VEL
LIN {X 0,Y 545.028,Z 363.222,A -85,B 0,C 180,E1 -3746.326,E2 -3746.326} C_VEL
LIN {X 0,Y 545.038,Z 363.213,A -85,B 0,C 180,E1 -3748.951,E2 -3748.951} C_VEL
LIN {X 0,Y 545.016,Z 363.216,A -85,B 0,C 180,E1 -3751.503,E2 -3751.503} C_VEL
LIN {X 0,Y 545.02,Z 363.222,A -85,B 0,C 180,E1 -3754.504,E2 -3754.504} C_VEL
LIN {X 0,Y 544.975,Z 363.221,A -85,B 0,C 180,E1 -3757.24,E2 -3757.24} C_VEL
LIN {X 0,Y 545.043,Z 363.219,A -85,B 0,C 180,E1 -3760.264,E2 -3760.264} C_VEL
LIN {X 0,Y 545.013,Z 363.22,A -85,B 0,C 180,E1 -3762.747,E2 -3762.747} C_VEL
LIN {X 0,Y 545.042,Z 363.213,A -85,B 0,C 180,E1 -3765.819,E2 -3765.819} C_VEL
LIN {X 0,Y 545.093,Z 363.208,A -85,B 0,C 180,E1 -3768.849,E2 -3768.849} C_VEL
LIN {X 0,Y 545.066,Z 363.21,A -85,B 0,C 180,E1 -3771.846,E2 -3771.846} C_VEL
LIN {X 0,Y 545.148,Z 363.204,A -85,B 0,C 180,E1 -3774.823,E2 -3774.823} C_VEL
LIN {X 0,Y 545.162,Z 363.195,A -85,B 0,C 180,E1 -3777.784,E2 -3777.784} C_VEL
LIN {X 0,Y 545.195,Z 363.199,A -85,B 0,C 180,E1 -3780.739,E2 -3780.739} C_VEL
LIN {X 0,Y 545.141,Z 363.204,A -85,B 0,C 180,E1 -3782.956,E2 -3782.956} C_VEL
LIN {X 0,Y 545.112,Z 363.2,A -85,B 0,C 180,E1 -3785.92,E2 -3785.92} C_VEL
LIN {X 0,Y 545.051,Z 363.207,A -85,B 0,C 180,E1 -3788.154,E2 -3788.154} C_VEL
LIN {X 0,Y 545.096,Z 363.208,A -85,B 0,C 180,E1 -3791.151,E2 -3791.151} C_VEL
LIN {X 0,Y 545.065,Z 363.206,A -85,B 0,C 180,E1 -3794.181,E2 -3794.181} C_VEL
LIN {X 0,Y 545.058,Z 363.211,A -85,B 0,C 180,E1 -3797.421,E2 -3797.421} C_VEL
LIN {X 0,Y 545.077,Z 363.208,A -85,B 0,C 180,E1 -3800.373,E2 -3800.373} C_VEL
LIN {X 0,Y 545.058,Z 363.211,A -85,B 0,C 180,E1 -3803.561,E2 -3803.561} C_VEL
LIN {X 0,Y 545.024,Z 363.212,A -85,B 0,C 180,E1 -3806.004,E2 -3806.004} C_VEL
LIN {X 0,Y 545.052,Z 363.218,A -85,B 0,C 180,E1 -3808.744,E2 -3808.744} C_VEL
LIN {X 0,Y 545.046,Z 363.208,A -85,B 0,C 180,E1 -3811.68,E2 -3811.68} C_VEL
LIN {X 0,Y 545.048,Z 363.217,A -85,B 0,C 180,E1 -3814.566,E2 -3814.566} C_VEL
LIN {X 0,Y 545.048,Z 363.217,A -85,B 0,C 180,E1 -3817.021,E2 -3817.021} C_VEL
LIN {X 0,Y 544.341,Z 363.303,A -85,B 0,C 180,E1 -3817.638,E2 -3817.638} C_VEL
LIN {X 0,Y 541.475,Z 363.662,A -85,B 0,C 180,E1 -3818.639,E2 -3818.639} C_VEL
LIN {X 0,Y 539.08,Z 363.956,A -85,B 0,C 180,E1 -3819.444,E2 -3819.444} C_VEL
LIN {X 0,Y 538.06,Z 364.081,A -85,B 0,C 180,E1 -3820.066,E2 -3820.066} C_VEL
LIN {X 0,Y 537.979,Z 364.092,A -85,B 0,C 180,E1 -3820.277,E2 -3820.277} C_VEL
LIN {X 0,Y 537.972,Z 364.1,A -85,B 0,C 180,E1 -3822.983,E2 -3822.983} C_VEL
LIN {X 0,Y 538.011,Z 364.088,A -85,B 0,C 180,E1 -3825.928,E2 -3825.928} C_VEL
LIN {X 0,Y 537.996,Z 364.095,A -85,B 0,C 180,E1 -3829.221,E2 -3829.221} C_VEL
LIN {X 0,Y 537.982,Z 364.091,A -85,B 0,C 180,E1 -3832.123,E2 -3832.123} C_VEL
LIN {X 0,Y 537.983,Z 364.098,A -85,B 0,C 180,E1 -3834.916,E2 -3834.916} C_VEL
LIN {X 0,Y 538.008,Z 364.092,A -85,B 0,C 180,E1 -3837.618,E2 -3837.618} C_VEL
LIN {X 0,Y 538.015,Z 364.18,A -85,B 0,C 180,E1 -3840.566,E2 -3840.566} C_VEL
LIN {X 0,Y 539.886,Z 369.129,A -85,B 0,C 180,E1 -3840.713,E2 -3840.713} C_VEL
LIN {X 0,Y 541.694,Z 373.418,A -85,B 0,C 180,E1 -3840.848,E2 -3840.848} C_VEL
LIN {X 0,Y 541.093,Z 492.356,A -85,B 0,C 180,E1 -3842.491,E2 -3842.491} C_VEL
LIN {X 0,Y 540.921,Z 507.681,A -85,B 0,C 180,E1 -3842.848,E2 -3842.848} C_VEL
LIN {X 0,Y 540.601,Z 522.594,A -85,B 0,C 180,E1 -3843.353,E2 -3843.353} C_VEL
LIN {X 0,Y 540.227,Z 537.572,A -85,B 0,C 180,E1 -3844.034,E2 -3844.034} C_VEL
LIN {X 0,Y 539.802,Z 551.836,A -85,B 0,C 180,E1 -3844.865,E2 -3844.865} C_VEL
LIN {X 0,Y 539.391,Z 564.687,A -85,B 0,C 180,E1 -3845.793,E2 -3845.793} C_VEL
LIN {X 0,Y 538.937,Z 576.974,A -85,B 0,C 180,E1 -3846.869,E2 -3846.869} C_VEL
LIN {X 0,Y 538.571,Z 587.779,A -85,B 0,C 180,E1 -3848.007,E2 -3848.007} C_VEL
LIN {X 0,Y 538.245,Z 598.428,A -85,B 0,C 180,E1 -3849.358,E2 -3849.358} C_VEL
LIN {X 0,Y 537.906,Z 608.705,A -85,B 0,C 180,E1 -3850.936,E2 -3850.936} C_VEL
LIN {X 0,Y 537.818,Z 615.237,A -85,B 0,C 180,E1 -3852.117,E2 -3852.117} C_VEL
LIN {X 0,Y 537.653,Z 622.303,A -85,B 0,C 180,E1 -3853.678,E2 -3853.678} C_VEL
LIN {X 0,Y 537.616,Z 626.515,A -85,B 0,C 180,E1 -3854.845,E2 -3854.845} C_VEL
LIN {X 0,Y 537.521,Z 630.915,A -85,B 0,C 180,E1 -3856.389,E2 -3856.389} C_VEL
LIN {X 0,Y 537.472,Z 633.996,A -85,B 0,C 180,E1 -3857.924,E2 -3857.924} C_VEL
LIN {X 0,Y 537.488,Z 635.847,A -85,B 0,C 180,E1 -3859.453,E2 -3859.453} C_VEL
LIN {X 0,Y 537.457,Z 636.491,A -85,B 0,C 180,E1 -3860.973,E2 -3860.973} C_VEL
LIN {X 0,Y 537.515,Z 635.945,A -85,B 0,C 180,E1 -3862.488,E2 -3862.488} C_VEL
LIN {X 0,Y 537.546,Z 634.253,A -85,B 0,C 180,E1 -3863.997,E2 -3863.997} C_VEL
LIN {X 0,Y 537.501,Z 631.394,A -85,B 0,C 180,E1 -3865.501,E2 -3865.501} C_VEL
LIN {X 0,Y 537.605,Z 627.311,A -85,B 0,C 180,E1 -3867.003,E2 -3867.003} C_VEL
LIN {X 0,Y 537.586,Z 621.934,A -85,B 0,C 180,E1 -3868.502,E2 -3868.502} C_VEL
LIN {X 0,Y 537.79,Z 615.105,A -85,B 0,C 180,E1 -3870,E2 -3870} C_VEL
LIN {X 0,Y 537.996,Z 606.637,A -85,B 0,C 180,E1 -3871.497,E2 -3871.497} C_VEL
LIN {X 0,Y 538.276,Z 596.477,A -85,B 0,C 180,E1 -3872.994,E2 -3872.994} C_VEL
LIN {X 0,Y 538.623,Z 587.442,A -85,B 0,C 180,E1 -3874.116,E2 -3874.116} C_VEL
LIN {X 0,Y 538.964,Z 576.749,A -85,B 0,C 180,E1 -3875.237,E2 -3875.237} C_VEL
LIN {X 0,Y 539.372,Z 565.016,A -85,B 0,C 180,E1 -3876.265,E2 -3876.265} C_VEL
LIN {X 0,Y 539.81,Z 552.14,A -85,B 0,C 180,E1 -3877.199,E2 -3877.199} C_VEL
LIN {X 0,Y 540.206,Z 538.841,A -85,B 0,C 180,E1 -3877.984,E2 -3877.984} C_VEL
LIN {X 0,Y 540.57,Z 524.539,A -85,B 0,C 180,E1 -3878.654,E2 -3878.654} C_VEL
LIN {X 0,Y 540.839,Z 509.337,A -85,B 0,C 180,E1 -3879.192,E2 -3879.192} C_VEL
LIN {X 0,Y 541.03,Z 493.418,A -85,B 0,C 180,E1 -3879.58,E2 -3879.58} C_VEL
LIN {X 0,Y 541.612,Z 373.085,A -85,B 0,C 180,E1 -3881.249,E2 -3881.249} C_VEL
LIN {X 0,Y 538.169,Z 364.673,A -85,B 0,C 180,E1 -3881.509,E2 -3881.509} C_VEL
LIN {X 0,Y 538.07,Z 364.087,A -85,B 0,C 180,E1 -3881.524,E2 -3881.524} C_VEL
LIN {X 0,Y 538.007,Z 364.097,A -85,B 0,C 180,E1 -3884.835,E2 -3884.835} C_VEL
LIN {X 0,Y 538.015,Z 364.09,A -85,B 0,C 180,E1 -3887.524,E2 -3887.524} C_VEL
LIN {X 0,Y 537.988,Z 364.095,A -85,B 0,C 180,E1 -3890.653,E2 -3890.653} C_VEL
LIN {X 0,Y 537.973,Z 364.101,A -85,B 0,C 180,E1 -3893.073,E2 -3893.073} C_VEL
LIN {X 0,Y 537.976,Z 364.095,A -85,B 0,C 180,E1 -3895.657,E2 -3895.657} C_VEL
LIN {X 0,Y 537.97,Z 364.094,A -85,B 0,C 180,E1 -3898.053,E2 -3898.053} C_VEL
LIN {X 0,Y 537.986,Z 364.089,A -85,B 0,C 180,E1 -3900.628,E2 -3900.628} C_VEL
LIN {X 0,Y 537.997,Z 364.096,A -85,B 0,C 180,E1 -3903.274,E2 -3903.274} C_VEL
LIN {X 0,Y 537.951,Z 364.095,A -85,B 0,C 180,E1 -3906.007,E2 -3906.007} C_VEL
LIN {X 0,Y 537.982,Z 364.096,A -85,B 0,C 180,E1 -3908.832,E2 -3908.832} C_VEL
LIN {X 0,Y 537.973,Z 364.093,A -85,B 0,C 180,E1 -3911.871,E2 -3911.871} C_VEL
LIN {X 0,Y 537.984,Z 364.095,A -85,B 0,C 180,E1 -3914.864,E2 -3914.864} C_VEL
LIN {X 0,Y 537.965,Z 364.101,A -85,B 0,C 180,E1 -3917.208,E2 -3917.208} C_VEL
LIN {X 0,Y 537.987,Z 364.091,A -85,B 0,C 180,E1 -3920.2,E2 -3920.2} C_VEL
LIN {X 0,Y 537.981,Z 364.097,A -85,B 0,C 180,E1 -3923.063,E2 -3923.063} C_VEL
LIN {X 0,Y 537.984,Z 364.091,A -85,B 0,C 180,E1 -3925.824,E2 -3925.824} C_VEL
LIN {X 0,Y 537.981,Z 364.092,A -85,B 0,C 180,E1 -3928.496,E2 -3928.496} C_VEL
LIN {X 0,Y 537.976,Z 364.097,A -85,B 0,C 180,E1 -3931.095,E2 -3931.095} C_VEL
LIN {X 0,Y 537.959,Z 364.099,A -85,B 0,C 180,E1 -3933.629,E2 -3933.629} C_VEL
LIN {X 0,Y 537.997,Z 364.088,A -85,B 0,C 180,E1 -3936.122,E2 -3936.122} C_VEL
LIN {X 0,Y 538.023,Z 364.096,A -85,B 0,C 180,E1 -3939.348,E2 -3939.348} C_VEL
LIN {X 0,Y 538.019,Z 364.086,A -85,B 0,C 180,E1 -3942.516,E2 -3942.516} C_VEL
LIN {X 0,Y 538.031,Z 364.089,A -85,B 0,C 180,E1 -3945.63,E2 -3945.63} C_VEL
LIN {X 0,Y 538.06,Z 364.073,A -85,B 0,C 180,E1 -3948.701,E2 -3948.701} C_VEL
LIN {X 0,Y 538.021,Z 364.09,A -85,B 0,C 180,E1 -3951.738,E2 -3951.738} C_VEL
LIN {X 0,Y 538.116,Z 364.075,A -85,B 0,C 180,E1 -3954.754,E2 -3954.754} C_VEL
LIN {X 0,Y 538.141,Z 364.075,A -85,B 0,C 180,E1 -3957.754,E2 -3957.754} C_VEL
LIN {X 0,Y 538.136,Z 364.075,A -85,B 0,C 180,E1 -3960,E2 -3960} C_VEL
LIN {X 0,Y 538.108,Z 364.076,A -85,B 0,C 180,E1 -3962.994,E2 -3962.994} C_VEL
LIN {X 0,Y 538.058,Z 364.085,A -85,B 0,C 180,E1 -3965.998,E2 -3965.998} C_VEL
LIN {X 0,Y 538.009,Z 364.088,A -85,B 0,C 180,E1 -3969.018,E2 -3969.018} C_VEL
LIN {X 0,Y 538.038,Z 364.087,A -85,B 0,C 180,E1 -3972.063,E2 -3972.063} C_VEL
LIN {X 0,Y 538.024,Z 364.086,A -85,B 0,C 180,E1 -3975.144,E2 -3975.144} C_VEL
LIN {X 0,Y 537.984,Z 364.091,A -85,B 0,C 180,E1 -3978.272,E2 -3978.272} C_VEL
LIN {X 0,Y 537.976,Z 364.092,A -85,B 0,C 180,E1 -3980.654,E2 -3980.654} C_VEL
LIN {X 0,Y 537.968,Z 364.093,A -85,B 0,C 180,E1 -3983.074,E2 -3983.074} C_VEL
LIN {X 0,Y 537.984,Z 364.1,A -85,B 0,C 180,E1 -3985.661,E2 -3985.661} C_VEL
LIN {X 0,Y 537.961,Z 364.099,A -85,B 0,C 180,E1 -3988.054,E2 -3988.054} C_VEL
LIN {X 0,Y 537.992,Z 364.091,A -85,B 0,C 180,E1 -3990.629,E2 -3990.629} C_VEL
LIN {X 0,Y 538.011,Z 364.089,A -85,B 0,C 180,E1 -3993.279,E2 -3993.279} C_VEL
LIN {X 0,Y 537.947,Z 364.103,A -85,B 0,C 180,E1 -3996.008,E2 -3996.008} C_VEL
LIN {X 0,Y 537.98,Z 364.089,A -85,B 0,C 180,E1 -3998.833,E2 -3998.833} C_VEL
LIN {X 0,Y 537.971,Z 364.099,A -85,B 0,C 180,E1 -4001.873,E2 -4001.873} C_VEL
LIN {X 0,Y 537.982,Z 364.091,A -85,B 0,C 180,E1 -4004.865,E2 -4004.865} C_VEL
LIN {X 0,Y 537.967,Z 364.096,A -85,B 0,C 180,E1 -4007.21,E2 -4007.21} C_VEL
LIN {X 0,Y 537.986,Z 364.094,A -85,B 0,C 180,E1 -4010.421,E2 -4010.421} C_VEL
LIN {X 0,Y 537.951,Z 364.097,A -85,B 0,C 180,E1 -4013.062,E2 -4013.062} C_VEL
LIN {X 0,Y 537.991,Z 364.099,A -85,B 0,C 180,E1 -4015.825,E2 -4015.825} C_VEL
LIN {X 0,Y 538.027,Z 364.232,A -85,B 0,C 180,E1 -4018.167,E2 -4018.167} C_VEL
LIN {X 0,Y 541.68,Z 378.376,A -85,B 0,C 180,E1 -4019.818,E2 -4019.818} C_VEL
LIN {X 0,Y 541.287,Z 403.364,A -85,B 0,C 180,E1 -4022.344,E2 -4022.344} C_VEL
LIN {X 0,Y 540.755,Z 431.404,A -85,B 0,C 180,E1 -4025.117,E2 -4025.117} C_VEL
LIN {X 0,Y 540.204,Z 462.56,A -85,B 0,C 180,E1 -4028.136,E2 -4028.136} C_VEL
LIN {X 0,Y 540.075,Z 472.662,A -85,B 0,C 180,E1 -4029.086,E2 -4029.086} C_VEL
LIN {X 0,Y 541.846,Z 484.446,A -85,B 0,C 180,E1 -4029.317,E2 -4029.317} C_VEL
LIN {X 0,Y 541.02,Z 640.751,A -85,B 0,C 180,E1 -4031.45,E2 -4031.45} C_VEL
LIN {X 0,Y 540.754,Z 656.706,A -85,B 0,C 180,E1 -4031.825,E2 -4031.825} C_VEL
LIN {X 0,Y 540.445,Z 672.036,A -85,B 0,C 180,E1 -4032.353,E2 -4032.353} C_VEL
LIN {X 0,Y 540.126,Z 685.785,A -85,B 0,C 180,E1 -4032.977,E2 -4032.977} C_VEL
LIN {X 0,Y 539.687,Z 699.256,A -85,B 0,C 180,E1 -4033.741,E2 -4033.741} C_VEL
LIN {X 0,Y 539.322,Z 712.237,A -85,B 0,C 180,E1 -4034.645,E2 -4034.645} C_VEL
LIN {X 0,Y 538.892,Z 724.29,A -85,B 0,C 180,E1 -4035.653,E2 -4035.653} C_VEL
LIN {X 0,Y 538.593,Z 735.748,A -85,B 0,C 180,E1 -4036.8,E2 -4036.8} C_VEL
LIN {X 0,Y 538.283,Z 745.388,A -85,B 0,C 180,E1 -4037.942,E2 -4037.942} C_VEL
LIN {X 0,Y 538.068,Z 754.854,A -85,B 0,C 180,E1 -4039.273,E2 -4039.273} C_VEL
LIN {X 0,Y 537.825,Z 762.734,A -85,B 0,C 180,E1 -4040.599,E2 -4040.599} C_VEL
LIN {X 0,Y 537.699,Z 770.089,A -85,B 0,C 180,E1 -4042.112,E2 -4042.112} C_VEL
LIN {X 0,Y 537.622,Z 775.405,A -85,B 0,C 180,E1 -4043.464,E2 -4043.464} C_VEL
LIN {X 0,Y 537.574,Z 779.386,A -85,B 0,C 180,E1 -4044.749,E2 -4044.749} C_VEL
LIN {X 0,Y 537.562,Z 782.887,A -85,B 0,C 180,E1 -4046.252,E2 -4046.252} C_VEL
LIN {X 0,Y 537.486,Z 785.19,A -85,B 0,C 180,E1 -4047.752,E2 -4047.752} C_VEL
LIN {X 0,Y 537.439,Z 786.348,A -85,B 0,C 180,E1 -4049.25,E2 -4049.25} C_VEL
LIN {X 0,Y 537.439,Z 786.347,A -85,B 0,C 180,E1 -4050.749,E2 -4050.749} C_VEL
LIN {X 0,Y 537.486,Z 785.187,A -85,B 0,C 180,E1 -4052.248,E2 -4052.248} C_VEL
LIN {X 0,Y 537.561,Z 782.885,A -85,B 0,C 180,E1 -4053.748,E2 -4053.748} C_VEL
LIN {X 0,Y 537.574,Z 779.388,A -85,B 0,C 180,E1 -4055.25,E2 -4055.25} C_VEL
LIN {X 0,Y 537.617,Z 774.611,A -85,B 0,C 180,E1 -4056.756,E2 -4056.756} C_VEL
LIN {X 0,Y 537.734,Z 768.423,A -85,B 0,C 180,E1 -4058.265,E2 -4058.265} C_VEL
LIN {X 0,Y 537.859,Z 760.647,A -85,B 0,C 180,E1 -4059.779,E2 -4059.779} C_VEL
LIN {X 0,Y 538.101,Z 752.371,A -85,B 0,C 180,E1 -4061.107,E2 -4061.107} C_VEL
LIN {X 0,Y 538.357,Z 742.396,A -85,B 0,C 180,E1 -4062.438,E2 -4062.438} C_VEL
LIN {X 0,Y 538.661,Z 732.191,A -85,B 0,C 180,E1 -4063.582,E2 -4063.582} C_VEL
LIN {X 0,Y 539.02,Z 720.026,A -85,B 0,C 180,E1 -4064.728,E2 -4064.728} C_VEL
LIN {X 0,Y 539.468,Z 707.835,A -85,B 0,C 180,E1 -4065.681,E2 -4065.681} C_VEL
LIN {X 0,Y 539.842,Z 694.516,A -85,B 0,C 180,E1 -4066.545,E2 -4066.545} C_VEL
LIN {X 0,Y 540.226,Z 679.836,A -85,B 0,C 180,E1 -4067.312,E2 -4067.312} C_VEL
LIN {X 0,Y 540.58,Z 664.327,A -85,B 0,C 180,E1 -4067.935,E2 -4067.935} C_VEL
LIN {X 0,Y 540.913,Z 648.77,A -85,B 0,C 180,E1 -4068.382,E2 -4068.382} C_VEL
LIN {X 0,Y 541.086,Z 633.243,A -85,B 0,C 180,E1 -4068.669,E2 -4068.669} C_VEL
LIN {X 0,Y 541.807,Z 483.023,A -85,B 0,C 180,E1 -4070.704,E2 -4070.704} C_VEL
LIN {X 0,Y 540.042,Z 472.17,A -85,B 0,C 180,E1 -4070.935,E2 -4070.935} C_VEL
LIN {X 0,Y 540.472,Z 443.73,A -85,B 0,C 180,E1 -4073.67,E2 -4073.67} C_VEL
LIN {X 0,Y 541.069,Z 415.087,A -85,B 0,C 180,E1 -4076.471,E2 -4076.471} C_VEL
LIN {X 0,Y 541.598,Z 384.356,A -85,B 0,C 180,E1 -4079.544,E2 -4079.544} C_VEL
LIN {X 0,Y 541.602,Z 378.061,A -85,B 0,C 180,E1 -4080.186,E2 -4080.186} C_VEL
LIN {X 0,Y 538.01,Z 364.098,A -85,B 0,C 180,E1 -4081.819,E2 -4081.819} C_VEL
LIN {X 0,Y 537.987,Z 364.095,A -85,B 0,C 180,E1 -4084.614,E2 -4084.614} C_VEL
LIN {X 0,Y 537.971,Z 364.1,A -85,B 0,C 180,E1 -4087.878,E2 -4087.878} C_VEL
LIN {X 0,Y 537.989,Z 364.092,A -85,B 0,C 180,E1 -4090.78,E2 -4090.78} C_VEL
LIN {X 0,Y 537.99,Z 364.099,A -85,B 0,C 180,E1 -4094.07,E2 -4094.07} C_VEL
LIN {X 0,Y 537.942,Z 364.096,A -85,B 0,C 180,E1 -4097.02,E2 -4097.02} C_VEL
LIN {X 0,Y 537.989,Z 364.09,A -85,B 0,C 180,E1 -4099.258,E2 -4099.258} C_VEL
LIN {X 0,Y 537.965,Z 364.1,A -85,B 0,C 180,E1 -4102.12,E2 -4102.12} C_VEL
LIN {X 0,Y 537.981,Z 364.092,A -85,B 0,C 180,E1 -4105.385,E2 -4105.385} C_VEL
LIN {X 0,Y 537.982,Z 364.099,A -85,B 0,C 180,E1 -4108.115,E2 -4108.115} C_VEL
LIN {X 0,Y 537.97,Z 364.094,A -85,B 0,C 180,E1 -4111.095,E2 -4111.095} C_VEL
LIN {X 0,Y 537.969,Z 364.094,A -85,B 0,C 180,E1 -4113.63,E2 -4113.63} C_VEL
LIN {X 0,Y 537.969,Z 364.099,A -85,B 0,C 180,E1 -4116.127,E2 -4116.127} C_VEL
LIN {X 0,Y 537.973,Z 364.099,A -85,B 0,C 180,E1 -4118.544,E2 -4118.544} C_VEL
LIN {X 0,Y 537.969,Z 364.096,A -85,B 0,C 180,E1 -4120.938,E2 -4120.938} C_VEL
LIN {X 0,Y 537.952,Z 364.095,A -85,B 0,C 180,E1 -4123.297,E2 -4123.297} C_VEL
LIN {X 0,Y 538.017,Z 364.087,A -85,B 0,C 180,E1 -4125.63,E2 -4125.63} C_VEL
LIN {X 0,Y 538.054,Z 364.087,A -85,B 0,C 180,E1 -4128.701,E2 -4128.701} C_VEL
LIN {X 0,Y 538.03,Z 364.086,A -85,B 0,C 180,E1 -4131.739,E2 -4131.739} C_VEL
LIN {X 0,Y 538.106,Z 364.082,A -85,B 0,C 180,E1 -4134.755,E2 -4134.755} C_VEL
LIN {X 0,Y 538.135,Z 364.07,A -85,B 0,C 180,E1 -4137.755,E2 -4137.755} C_VEL
LIN {X 0,Y 538.164,Z 364.074,A -85,B 0,C 180,E1 -4140.748,E2 -4140.748} C_VEL
LIN {X 0,Y 538.106,Z 364.08,A -85,B 0,C 180,E1 -4142.995,E2 -4142.995} C_VEL
LIN {X 0,Y 538.069,Z 364.078,A -85,B 0,C 180,E1 -4145.998,E2 -4145.998} C_VEL
LIN {X 0,Y 538.023,Z 364.083,A -85,B 0,C 180,E1 -4148.262,E2 -4148.262} C_VEL
LIN {X 0,Y 538.068,Z 364.08,A -85,B 0,C 180,E1 -4151.597,E2 -4151.597} C_VEL
LIN {X 0,Y 538.033,Z 364.087,A -85,B 0,C 180,E1 -4154.853,E2 -4154.853} C_VEL
LIN {X 0,Y 538.022,Z 364.087,A -85,B 0,C 180,E1 -4157.533,E2 -4157.533} C_VEL
LIN {X 0,Y 538.022,Z 364.089,A -85,B 0,C 180,E1 -4160.652,E2 -4160.652} C_VEL
LIN {X 0,Y 537.993,Z 364.09,A -85,B 0,C 180,E1 -4163.878,E2 -4163.878} C_VEL
LIN {X 0,Y 537.968,Z 364.094,A -85,B 0,C 180,E1 -4166.371,E2 -4166.371} C_VEL
LIN {X 0,Y 538.018,Z 364.096,A -85,B 0,C 180,E1 -4168.934,E2 -4168.934} C_VEL
LIN {X 0,Y 537.998,Z 364.086,A -85,B 0,C 180,E1 -4171.888,E2 -4171.888} C_VEL
LIN {X 0,Y 537.998,Z 364.096,A -85,B 0,C 180,E1 -4174.618,E2 -4174.618} C_VEL
LIN {X 0,Y 537.993,Z 364.096,A -85,B 0,C 180,E1 -4177.171,E2 -4177.171} C_VEL
LIN {X 0,Y 537.999,Z 364.089,A -85,B 0,C 180,E1 -4179.799,E2 -4179.799} C_VEL
LIN {X 0,Y 537.979,Z 364.092,A -85,B 0,C 180,E1 -4180.277,E2 -4180.277} C_VEL
LIN {X 0,Y 537.319,Z 364.18,A -85,B 0,C 180,E1 -4180.902,E2 -4180.902} C_VEL
LIN {X 0,Y 534.467,Z 364.535,A -85,B 0,C 180,E1 -4181.917,E2 -4181.917} C_VEL
LIN {X 0,Y 532.051,Z 364.837,A -85,B 0,C 180,E1 -4182.734,E2 -4182.734} C_VEL
LIN {X 0,Y 531.012,Z 364.961,A -85,B 0,C 180,E1 -4183.365,E2 -4183.365} C_VEL
LIN {X 0,Y 530.927,Z 364.969,A -85,B 0,C 180,E1 -4183.579,E2 -4183.579} C_VEL
LIN {X 0,Y 530.938,Z 364.972,A -85,B 0,C 180,E1 -4186.504,E2 -4186.504} C_VEL
LIN {X 0,Y 530.944,Z 364.97,A -85,B 0,C 180,E1 -4189.565,E2 -4189.565} C_VEL
LIN {X 0,Y 530.96,Z 364.968,A -85,B 0,C 180,E1 -4192.579,E2 -4192.579} C_VEL
LIN {X 0,Y 530.965,Z 364.974,A -85,B 0,C 180,E1 -4195.31,E2 -4195.31} C_VEL
LIN {X 0,Y 530.954,Z 364.968,A -85,B 0,C 180,E1 -4198.032,E2 -4198.032} C_VEL
LIN {X 0,Y 530.97,Z 364.969,A -85,B 0,C 180,E1 -4200.265,E2 -4200.265} C_VEL
LIN {X 0,Y 532.467,Z 369.081,A -85,B 0,C 180,E1 -4200.4,E2 -4200.4} C_VEL
LIN {X 0,Y 535.044,Z 375.117,A -85,B 0,C 180,E1 -4200.595,E2 -4200.595} C_VEL
LIN {X 0,Y 534.423,Z 492.504,A -85,B 0,C 180,E1 -4202.237,E2 -4202.237} C_VEL
LIN {X 0,Y 534.252,Z 507.744,A -85,B 0,C 180,E1 -4202.587,E2 -4202.587} C_VEL
LIN {X 0,Y 533.906,Z 522.942,A -85,B 0,C 180,E1 -4203.098,E2 -4203.098} C_VEL
LIN {X 0,Y 533.589,Z 536.731,A -85,B 0,C 180,E1 -4203.721,E2 -4203.721} C_VEL
LIN {X 0,Y 533.167,Z 549.221,A -85,B 0,C 180,E1 -4204.426,E2 -4204.426} C_VEL
LIN {X 0,Y 532.712,Z 562.896,A -85,B 0,C 180,E1 -4205.377,E2 -4205.377} C_VEL
LIN {X 0,Y 532.292,Z 574.486,A -85,B 0,C 180,E1 -4206.357,E2 -4206.357} C_VEL
LIN {X 0,Y 531.872,Z 585.506,A -85,B 0,C 180,E1 -4207.469,E2 -4207.469} C_VEL
LIN {X 0,Y 531.445,Z 595.56,A -85,B 0,C 180,E1 -4208.675,E2 -4208.675} C_VEL
LIN {X 0,Y 531.181,Z 604.459,A -85,B 0,C 180,E1 -4209.951,E2 -4209.951} C_VEL
LIN {X 0,Y 530.907,Z 612.224,A -85,B 0,C 180,E1 -4211.277,E2 -4211.277} C_VEL
LIN {X 0,Y 530.7,Z 619.312,A -85,B 0,C 180,E1 -4212.752,E2 -4212.752} C_VEL
LIN {X 0,Y 530.539,Z 625.05,A -85,B 0,C 180,E1 -4214.244,E2 -4214.244} C_VEL
LIN {X 0,Y 530.504,Z 628.654,A -85,B 0,C 180,E1 -4215.422,E2 -4215.422} C_VEL
LIN {X 0,Y 530.39,Z 632.379,A -85,B 0,C 180,E1 -4216.982,E2 -4216.982} C_VEL
LIN {X 0,Y 530.448,Z 635.061,A -85,B 0,C 180,E1 -4218.65,E2 -4218.65} C_VEL
LIN {X 0,Y 530.385,Z 636.257,A -85,B 0,C 180,E1 -4220.081,E2 -4220.081} C_VEL
LIN {X 0,Y 530.414,Z 636.386,A -85,B 0,C 180,E1 -4221.62,E2 -4221.62} C_VEL
LIN {X 0,Y 530.466,Z 635.368,A -85,B 0,C 180,E1 -4223.152,E2 -4223.152} C_VEL
LIN {X 0,Y 530.456,Z 633.2,A -85,B 0,C 180,E1 -4224.679,E2 -4224.679} C_VEL
LIN {X 0,Y 530.501,Z 629.889,A -85,B 0,C 180,E1 -4226.202,E2 -4226.202} C_VEL
LIN {X 0,Y 530.482,Z 625.479,A -85,B 0,C 180,E1 -4227.723,E2 -4227.723} C_VEL
LIN {X 0,Y 530.639,Z 619.716,A -85,B 0,C 180,E1 -4229.241,E2 -4229.241} C_VEL
LIN {X 0,Y 530.915,Z 612.481,A -85,B 0,C 180,E1 -4230.759,E2 -4230.759} C_VEL
LIN {X 0,Y 531.147,Z 604.758,A -85,B 0,C 180,E1 -4232.086,E2 -4232.086} C_VEL
LIN {X 0,Y 531.487,Z 595.515,A -85,B 0,C 180,E1 -4233.412,E2 -4233.412} C_VEL
LIN {X 0,Y 531.851,Z 586.092,A -85,B 0,C 180,E1 -4234.548,E2 -4234.548} C_VEL
LIN {X 0,Y 532.273,Z 574.926,A -85,B 0,C 180,E1 -4235.683,E2 -4235.683} C_VEL
LIN {X 0,Y 532.7,Z 562.646,A -85,B 0,C 180,E1 -4236.724,E2 -4236.724} C_VEL
LIN {X 0,Y 533.204,Z 549.006,A -85,B 0,C 180,E1 -4237.669,E2 -4237.669} C_VEL
LIN {X 0,Y 533.588,Z 535.164,A -85,B 0,C 180,E1 -4238.442,E2 -4238.442} C_VEL
LIN {X 0,Y 533.953,Z 521.517,A -85,B 0,C 180,E1 -4239.04,E2 -4239.04} C_VEL
LIN {X 0,Y 534.197,Z 506.43,A -85,B 0,C 180,E1 -4239.537,E2 -4239.537} C_VEL
LIN {X 0,Y 534.361,Z 491.572,A -85,B 0,C 180,E1 -4239.869,E2 -4239.869} C_VEL
LIN {X 0,Y 534.95,Z 374.798,A -85,B 0,C 180,E1 -4241.501,E2 -4241.501} C_VEL
LIN {X 0,Y 531.135,Z 365.599,A -85,B 0,C 180,E1 -4241.793,E2 -4241.793} C_VEL
LIN {X 0,Y 531.013,Z 364.964,A -85,B 0,C 180,E1 -4241.811,E2 -4241.811} C_VEL
LIN {X 0,Y 530.964,Z 364.974,A -85,B 0,C 180,E1 -4244.927,E2 -4244.927} C_VEL
LIN {X 0,Y 530.973,Z 364.966,A -85,B 0,C 180,E1 -4247.724,E2 -4247.724} C_VEL
LIN {X 0,Y 530.961,Z 364.974,A -85,B 0,C 180,E1 -4250.939,E2 -4250.939} C_VEL
LIN {X 0,Y 530.938,Z 364.97,A -85,B 0,C 180,E1 -4254.027,E2 -4254.027} C_VEL
LIN {X 0,Y 530.942,Z 364.974,A -85,B 0,C 180,E1 -4256.747,E2 -4256.747} C_VEL
LIN {X 0,Y 530.914,Z 364.973,A -85,B 0,C 180,E1 -4259.326,E2 -4259.326} C_VEL
LIN {X 0,Y 530.948,Z 364.968,A -85,B 0,C 180,E1 -4262.097,E2 -4262.097} C_VEL
LIN {X 0,Y 530.95,Z 364.972,A -85,B 0,C 180,E1 -4264.847,E2 -4264.847} C_VEL
LIN {X 0,Y 530.925,Z 364.975,A -85,B 0,C 180,E1 -4267.51,E2 -4267.51} C_VEL
LIN {X 0,Y 530.929,Z 364.969,A -85,B 0,C 180,E1 -4270.437,E2 -4270.437} C_VEL
LIN {X 0,Y 530.915,Z 364.975,A -85,B 0,C 180,E1 -4273.499,E2 -4273.499} C_VEL
LIN {X 0,Y 530.958,Z 364.97,A -85,B 0,C 180,E1 -4275.623,E2 -4275.623} C_VEL
LIN {X 0,Y 530.928,Z 364.975,A -85,B 0,C 180,E1 -4278.982,E2 -4278.982} C_VEL
LIN {X 0,Y 530.923,Z 364.975,A -85,B 0,C 180,E1 -4281.526,E2 -4281.526} C_VEL
LIN {X 0,Y 530.928,Z 364.971,A -85,B 0,C 180,E1 -4284.378,E2 -4284.378} C_VEL
LIN {X 0,Y 530.937,Z 364.974,A -85,B 0,C 180,E1 -4287.131,E2 -4287.131} C_VEL
LIN {X 0,Y 530.922,Z 364.972,A -85,B 0,C 180,E1 -4289.8,E2 -4289.8} C_VEL
LIN {X 0,Y 530.945,Z 364.968,A -85,B 0,C 180,E1 -4292.479,E2 -4292.479} C_VEL
LIN {X 0,Y 530.936,Z 364.97,A -85,B 0,C 180,E1 -4295.773,E2 -4295.773} C_VEL
LIN {X 0,Y 530.985,Z 364.968,A -85,B 0,C 180,E1 -4299.061,E2 -4299.061} C_VEL
LIN {X 0,Y 530.955,Z 364.973,A -85,B 0,C 180,E1 -4301.477,E2 -4301.477} C_VEL
LIN {X 0,Y 530.974,Z 364.965,A -85,B 0,C 180,E1 -4304.649,E2 -4304.649} C_VEL
LIN {X 0,Y 531.007,Z 364.954,A -85,B 0,C 180,E1 -4307.774,E2 -4307.774} C_VEL
LIN {X 0,Y 530.947,Z 364.96,A -85,B 0,C 180,E1 -4310.091,E2 -4310.091} C_VEL
LIN {X 0,Y 531.001,Z 364.963,A -85,B 0,C 180,E1 -4313.159,E2 -4313.159} C_VEL
LIN {X 0,Y 530.964,Z 364.975,A -85,B 0,C 180,E1 -4315.445,E2 -4315.445} C_VEL
LIN {X 0,Y 531.114,Z 364.95,A -85,B 0,C 180,E1 -4317.725,E2 -4317.725} C_VEL
LIN {X 0,Y 531.106,Z 364.95,A -85,B 0,C 180,E1 -4320,E2 -4320} C_VEL
LIN {X 0,Y 531.076,Z 364.952,A -85,B 0,C 180,E1 -4323.034,E2 -4323.034} C_VEL
LIN {X 0,Y 531.018,Z 364.961,A -85,B 0,C 180,E1 -4326.078,E2 -4326.078} C_VEL
LIN {X 0,Y 530.976,Z 364.965,A -85,B 0,C 180,E1 -4329.139,E2 -4329.139} C_VEL
LIN {X 0,Y 531.036,Z 364.966,A -85,B 0,C 180,E1 -4331.669,E2 -4331.669} C_VEL
LIN {X 0,Y 531.007,Z 364.959,A -85,B 0,C 180,E1 -4334.95,E2 -4334.95} C_VEL
LIN {X 0,Y 530.96,Z 364.973,A -85,B 0,C 180,E1 -4337.724,E2 -4337.724} C_VEL
LIN {X 0,Y 530.96,Z 364.969,A -85,B 0,C 180,E1 -4340.13,E2 -4340.13} C_VEL
LIN {X 0,Y 530.907,Z 364.971,A -85,B 0,C 180,E1 -4342.575,E2 -4342.575} C_VEL
LIN {X 0,Y 530.938,Z 364.97,A -85,B 0,C 180,E1 -4345.061,E2 -4345.061} C_VEL
LIN {X 0,Y 530.94,Z 364.975,A -85,B 0,C 180,E1 -4347.6,E2 -4347.6} C_VEL
LIN {X 0,Y 530.946,Z 364.969,A -85,B 0,C 180,E1 -4350.642,E2 -4350.642} C_VEL
LIN {X 0,Y 530.94,Z 364.973,A -85,B 0,C 180,E1 -4353.776,E2 -4353.776} C_VEL
LIN {X 0,Y 530.897,Z 364.975,A -85,B 0,C 180,E1 -4356.563,E2 -4356.563} C_VEL
LIN {X 0,Y 530.944,Z 364.969,A -85,B 0,C 180,E1 -4359.447,E2 -4359.447} C_VEL
LIN {X 0,Y 530.898,Z 364.974,A -85,B 0,C 180,E1 -4362.464,E2 -4362.464} C_VEL
LIN {X 0,Y 530.954,Z 364.97,A -85,B 0,C 180,E1 -4365.451,E2 -4365.451} C_VEL
LIN {X 0,Y 530.905,Z 364.97,A -85,B 0,C 180,E1 -4368.557,E2 -4368.557} C_VEL
LIN {X 0,Y 530.94,Z 364.973,A -85,B 0,C 180,E1 -4371.529,E2 -4371.529} C_VEL
LIN {X 0,Y 530.923,Z 364.977,A -85,B 0,C 180,E1 -4374.378,E2 -4374.378} C_VEL
LIN {X 0,Y 530.972,Z 364.972,A -85,B 0,C 180,E1 -4377.554,E2 -4377.554} C_VEL
LIN {X 0,Y 530.975,Z 365.107,A -85,B 0,C 180,E1 -4377.898,E2 -4377.898} C_VEL
LIN {X 0,Y 534.951,Z 380.553,A -85,B 0,C 180,E1 -4379.725,E2 -4379.725} C_VEL
LIN {X 0,Y 534.418,Z 405.518,A -85,B 0,C 180,E1 -4382.277,E2 -4382.277} C_VEL
LIN {X 0,Y 533.868,Z 431.447,A -85,B 0,C 180,E1 -4384.878,E2 -4384.878} C_VEL
LIN {X 0,Y 533.256,Z 462.573,A -85,B 0,C 180,E1 -4387.938,E2 -4387.938} C_VEL
LIN {X 0,Y 533.11,Z 471.544,A -85,B 0,C 180,E1 -4388.799,E2 -4388.799} C_VEL
LIN {X 0,Y 535.171,Z 484.864,A -85,B 0,C 180,E1 -4389.067,E2 -4389.067} C_VEL
LIN {X 0,Y 534.246,Z 640.697,A -85,B 0,C 180,E1 -4391.223,E2 -4391.223} C_VEL
LIN {X 0,Y 533.966,Z 656.735,A -85,B 0,C 180,E1 -4391.611,E2 -4391.611} C_VEL
LIN {X 0,Y 533.644,Z 671.484,A -85,B 0,C 180,E1 -4392.12,E2 -4392.12} C_VEL
LIN {X 0,Y 533.275,Z 685.451,A -85,B 0,C 180,E1 -4392.751,E2 -4392.751} C_VEL
LIN {X 0,Y 532.818,Z 699.172,A -85,B 0,C 180,E1 -4393.526,E2 -4393.526} C_VEL
LIN {X 0,Y 532.443,Z 711.673,A -85,B 0,C 180,E1 -4394.399,E2 -4394.399} C_VEL
LIN {X 0,Y 531.965,Z 724.288,A -85,B 0,C 180,E1 -4395.462,E2 -4395.462} C_VEL
LIN {X 0,Y 531.607,Z 735.747,A -85,B 0,C 180,E1 -4396.623,E2 -4396.623} C_VEL
LIN {X 0,Y 531.286,Z 745.388,A -85,B 0,C 180,E1 -4397.781,E2 -4397.781} C_VEL
LIN {X 0,Y 531.051,Z 754.853,A -85,B 0,C 180,E1 -4399.13,E2 -4399.13} C_VEL
LIN {X 0,Y 530.765,Z 762.734,A -85,B 0,C 180,E1 -4400.473,E2 -4400.473} C_VEL
LIN {X 0,Y 530.64,Z 770.089,A -85,B 0,C 180,E1 -4402.006,E2 -4402.006} C_VEL
LIN {X 0,Y 530.542,Z 775.707,A -85,B 0,C 180,E1 -4403.469,E2 -4403.469} C_VEL
LIN {X 0,Y 530.508,Z 779.386,A -85,B 0,C 180,E1 -4404.679,E2 -4404.679} C_VEL
LIN {X 0,Y 530.481,Z 782.887,A -85,B 0,C 180,E1 -4406.202,E2 -4406.202} C_VEL
LIN {X 0,Y 530.407,Z 785.189,A -85,B 0,C 180,E1 -4407.722,E2 -4407.722} C_VEL
LIN {X 0,Y 530.341,Z 786.348,A -85,B 0,C 180,E1 -4409.24,E2 -4409.24} C_VEL
LIN {X 0,Y 530.341,Z 786.347,A -85,B 0,C 180,E1 -4410.759,E2 -4410.759} C_VEL
LIN {X 0,Y 530.407,Z 785.187,A -85,B 0,C 180,E1 -4412.278,E2 -4412.278} C_VEL
LIN {X 0,Y 530.48,Z 782.884,A -85,B 0,C 180,E1 -4413.798,E2 -4413.798} C_VEL
LIN {X 0,Y 530.508,Z 779.388,A -85,B 0,C 180,E1 -4415.32,E2 -4415.32} C_VEL
LIN {X 0,Y 530.549,Z 774.611,A -85,B 0,C 180,E1 -4416.847,E2 -4416.847} C_VEL
LIN {X 0,Y 530.665,Z 768.422,A -85,B 0,C 180,E1 -4418.376,E2 -4418.376} C_VEL
LIN {X 0,Y 530.809,Z 760.646,A -85,B 0,C 180,E1 -4419.911,E2 -4419.911} C_VEL
LIN {X 0,Y 531.056,Z 752.37,A -85,B 0,C 180,E1 -4421.256,E2 -4421.256} C_VEL
LIN {X 0,Y 531.382,Z 742.396,A -85,B 0,C 180,E1 -4422.604,E2 -4422.604} C_VEL
LIN {X 0,Y 531.709,Z 732.19,A -85,B 0,C 180,E1 -4423.763,E2 -4423.763} C_VEL
LIN {X 0,Y 532.119,Z 720.025,A -85,B 0,C 180,E1 -4424.924,E2 -4424.924} C_VEL
LIN {X 0,Y 532.6,Z 706.598,A -85,B 0,C 180,E1 -4425.98,E2 -4425.98} C_VEL
LIN {X 0,Y 533.042,Z 692.686,A -85,B 0,C 180,E1 -4426.861,E2 -4426.861} C_VEL
LIN {X 0,Y 533.427,Z 678.342,A -85,B 0,C 180,E1 -4427.589,E2 -4427.589} C_VEL
LIN {X 0,Y 533.78,Z 663.629,A -85,B 0,C 180,E1 -4428.172,E2 -4428.172} C_VEL
LIN {X 0,Y 534.113,Z 647.994,A -85,B 0,C 180,E1 -4428.622,E2 -4428.622} C_VEL
LIN {X 0,Y 534.295,Z 631.464,A -85,B 0,C 180,E1 -4428.926,E2 -4428.926} C_VEL
LIN {X 0,Y 535.198,Z 484.824,A -85,B 0,C 180,E1 -4430.931,E2 -4430.931} C_VEL
LIN {X 0,Y 533.062,Z 471.14,A -85,B 0,C 180,E1 -4431.215,E2 -4431.215} C_VEL
LIN {X 0,Y 533.591,Z 442.659,A -85,B 0,C 180,E1 -4433.994,E2 -4433.994} C_VEL
LIN {X 0,Y 534.237,Z 414.631,A -85,B 0,C 180,E1 -4436.779,E2 -4436.779} C_VEL
LIN {X 0,Y 534.881,Z 384.195,A -85,B 0,C 180,E1 -4439.865,E2 -4439.865} C_VEL
LIN {X 0,Y 534.668,Z 379.144,A -85,B 0,C 180,E1 -4440.401,E2 -4440.401} C_VEL
LIN {X 0,Y 530.961,Z 364.976,A -85,B 0,C 180,E1 -4442.1,E2 -4442.1} C_VEL
LIN {X 0,Y 530.948,Z 364.97,A -85,B 0,C 180,E1 -4444.848,E2 -4444.848} C_VEL
LIN {X 0,Y 530.921,Z 364.974,A -85,B 0,C 180,E1 -4447.51,E2 -4447.51} C_VEL
LIN {X 0,Y 530.938,Z 364.974,A -85,B 0,C 180,E1 -4450.435,E2 -4450.435} C_VEL
LIN {X 0,Y 530.918,Z 364.973,A -85,B 0,C 180,E1 -4453.498,E2 -4453.498} C_VEL
LIN {X 0,Y 530.951,Z 364.965,A -85,B 0,C 180,E1 -4455.623,E2 -4455.623} C_VEL
LIN {X 0,Y 530.923,Z 364.971,A -85,B 0,C 180,E1 -4458.982,E2 -4458.982} C_VEL
LIN {X 0,Y 530.934,Z 364.969,A -85,B 0,C 180,E1 -4461.528,E2 -4461.528} C_VEL
LIN {X 0,Y 530.915,Z 364.98,A -85,B 0,C 180,E1 -4464.377,E2 -4464.377} C_VEL
LIN {X 0,Y 530.94,Z 364.969,A -85,B 0,C 180,E1 -4467.132,E2 -4467.132} C_VEL
LIN {X 0,Y 530.931,Z 364.971,A -85,B 0,C 180,E1 -4469.801,E2 -4469.801} C_VEL
LIN {X 0,Y 530.939,Z 364.976,A -85,B 0,C 180,E1 -4472.479,E2 -4472.479} C_VEL
LIN {X 0,Y 530.933,Z 364.971,A -85,B 0,C 180,E1 -4474.939,E2 -4474.939} C_VEL
LIN {X 0,Y 530.932,Z 364.979,A -85,B 0,C 180,E1 -4478.245,E2 -4478.245} C_VEL
LIN {X 0,Y 530.924,Z 364.977,A -85,B 0,C 180,E1 -4480.675,E2 -4480.675} C_VEL
LIN {X 0,Y 530.92,Z 364.972,A -85,B 0,C 180,E1 -4483.069,E2 -4483.069} C_VEL
LIN {X 0,Y 530.98,Z 364.964,A -85,B 0,C 180,E1 -4485.435,E2 -4485.435} C_VEL
LIN {X 0,Y 531.014,Z 364.967,A -85,B 0,C 180,E1 -4488.549,E2 -4488.549} C_VEL
LIN {X 0,Y 530.976,Z 364.965,A -85,B 0,C 180,E1 -4491.628,E2 -4491.628} C_VEL
LIN {X 0,Y 531.066,Z 364.96,A -85,B 0,C 180,E1 -4494.685,E2 -4494.685} C_VEL
LIN {X 0,Y 531.109,Z 364.945,A -85,B 0,C 180,E1 -4497.725,E2 -4497.725} C_VEL
LIN {X 0,Y 531.134,Z 364.949,A -85,B 0,C 180,E1 -4500.758,E2 -4500.758} C_VEL
LIN {X 0,Y 531.071,Z 364.955,A -85,B 0,C 180,E1 -4503.035,E2 -4503.035} C_VEL
LIN {X 0,Y 531.03,Z 364.955,A -85,B 0,C 180,E1 -4506.078,E2 -4506.078} C_VEL
LIN {X 0,Y 530.974,Z 364.962,A -85,B 0,C 180,E1 -4508.372,E2 -4508.372} C_VEL
LIN {X 0,Y 531.032,Z 364.957,A -85,B 0,C 180,E1 -4511.67,E2 -4511.67} C_VEL
LIN {X 0,Y 531.008,Z 364.963,A -85,B 0,C 180,E1 -4514.953,E2 -4514.953} C_VEL
LIN {X 0,Y 530.967,Z 364.965,A -85,B 0,C 180,E1 -4517.724,E2 -4517.724} C_VEL
LIN {X 0,Y 531.011,Z 364.958,A -85,B 0,C 180,E1 -4520.128,E2 -4520.128} C_VEL
LIN {X 0,Y 530.928,Z 364.972,A -85,B 0,C 180,E1 -4522.574,E2 -4522.574} C_VEL
LIN {X 0,Y 530.934,Z 364.972,A -85,B 0,C 180,E1 -4525.061,E2 -4525.061} C_VEL
LIN {X 0,Y 530.948,Z 364.966,A -85,B 0,C 180,E1 -4527.6,E2 -4527.6} C_VEL
LIN {X 0,Y 530.941,Z 364.971,A -85,B 0,C 180,E1 -4530.199,E2 -4530.199} C_VEL
LIN {X 0,Y 530.955,Z 364.972,A -85,B 0,C 180,E1 -4532.868,E2 -4532.868} C_VEL
LIN {X 0,Y 530.943,Z 364.968,A -85,B 0,C 180,E1 -4535.621,E2 -4535.621} C_VEL
LIN {X 0,Y 530.953,Z 364.973,A -85,B 0,C 180,E1 -4538.654,E2 -4538.654} C_VEL
LIN {X 0,Y 530.954,Z 364.97,A -85,B 0,C 180,E1 -4541.44,E2 -4541.44} C_VEL
LIN {X 0,Y 530.927,Z 364.969,A -85,B 0,C 180,E1 -4543.579,E2 -4543.579} C_VEL
LIN {X 0,Y 530.263,Z 365.051,A -85,B 0,C 180,E1 -4544.212,E2 -4544.212} C_VEL
LIN {X 0,Y 527.423,Z 365.413,A -85,B 0,C 180,E1 -4545.241,E2 -4545.241} C_VEL
LIN {X 0,Y 525.018,Z 365.716,A -85,B 0,C 180,E1 -4546.07,E2 -4546.07} C_VEL
LIN {X 0,Y 523.977,Z 365.843,A -85,B 0,C 180,E1 -4546.71,E2 -4546.71} C_VEL
LIN {X 0,Y 523.887,Z 365.852,A -85,B 0,C 180,E1 -4546.926,E2 -4546.926} C_VEL
LIN {X 0,Y 523.906,Z 365.845,A -85,B 0,C 180,E1 -4549.918,E2 -4549.918} C_VEL
LIN {X 0,Y 523.899,Z 365.851,A -85,B 0,C 180,E1 -4552.869,E2 -4552.869} C_VEL
LIN {X 0,Y 523.908,Z 365.848,A -85,B 0,C 180,E1 -4555.709,E2 -4555.709} C_VEL
LIN {X 0,Y 523.907,Z 365.848,A -85,B 0,C 180,E1 -4558.456,E2 -4558.456} C_VEL
LIN {X 0,Y 523.926,Z 365.847,A -85,B 0,C 180,E1 -4559.973,E2 -4559.973} C_VEL
LIN {X 0,Y 525.423,Z 369.953,A -85,B 0,C 180,E1 -4560.107,E2 -4560.107} C_VEL
LIN {X 0,Y 528.469,Z 377.092,A -85,B 0,C 180,E1 -4560.343,E2 -4560.343} C_VEL
LIN {X 0,Y 527.759,Z 493.931,A -85,B 0,C 180,E1 -4561.997,E2 -4561.997} C_VEL
LIN {X 0,Y 527.583,Z 508.769,A -85,B 0,C 180,E1 -4562.345,E2 -4562.345} C_VEL
LIN {X 0,Y 527.239,Z 523.296,A -85,B 0,C 180,E1 -4562.837,E2 -4562.837} C_VEL
LIN {X 0,Y 526.906,Z 537.238,A -85,B 0,C 180,E1 -4563.468,E2 -4563.468} C_VEL
LIN {X 0,Y 526.463,Z 549.847,A -85,B 0,C 180,E1 -4564.182,E2 -4564.182} C_VEL
LIN {X 0,Y 526,Z 562.916,A -85,B 0,C 180,E1 -4565.093,E2 -4565.093} C_VEL
LIN {X 0,Y 525.507,Z 575.246,A -85,B 0,C 180,E1 -4566.138,E2 -4566.138} C_VEL
LIN {X 0,Y 525.066,Z 586.432,A -85,B 0,C 180,E1 -4567.278,E2 -4567.278} C_VEL
LIN {X 0,Y 524.564,Z 597.153,A -85,B 0,C 180,E1 -4568.588,E2 -4568.588} C_VEL
LIN {X 0,Y 524.309,Z 605.277,A -85,B 0,C 180,E1 -4569.769,E2 -4569.769} C_VEL
LIN {X 0,Y 523.979,Z 613.636,A -85,B 0,C 180,E1 -4571.223,E2 -4571.223} C_VEL
LIN {X 0,Y 523.697,Z 621.109,A -85,B 0,C 180,E1 -4572.829,E2 -4572.829} C_VEL
LIN {X 0,Y 523.569,Z 626.967,A -85,B 0,C 180,E1 -4574.428,E2 -4574.428} C_VEL
LIN {X 0,Y 523.454,Z 631.402,A -85,B 0,C 180,E1 -4576.015,E2 -4576.015} C_VEL
LIN {X 0,Y 523.353,Z 634.547,A -85,B 0,C 180,E1 -4577.593,E2 -4577.593} C_VEL
LIN {X 0,Y 523.376,Z 636.451,A -85,B 0,C 180,E1 -4579.165,E2 -4579.165} C_VEL
LIN {X 0,Y 523.315,Z 637.229,A -85,B 0,C 180,E1 -4580.726,E2 -4580.726} C_VEL
LIN {X 0,Y 523.375,Z 636.888,A -85,B 0,C 180,E1 -4582.283,E2 -4582.283} C_VEL
LIN {X 0,Y 523.416,Z 635.458,A -85,B 0,C 180,E1 -4583.834,E2 -4583.834} C_VEL
LIN {X 0,Y 523.399,Z 632.929,A -85,B 0,C 180,E1 -4585.379,E2 -4585.379} C_VEL
LIN {X 0,Y 523.555,Z 629.171,A -85,B 0,C 180,E1 -4586.922,E2 -4586.922} C_VEL
LIN {X 0,Y 523.541,Z 624.2,A -85,B 0,C 180,E1 -4588.462,E2 -4588.462} C_VEL
LIN {X 0,Y 523.792,Z 617.83,A -85,B 0,C 180,E1 -4590,E2 -4590} C_VEL
LIN {X 0,Y 524.113,Z 609.915,A -85,B 0,C 180,E1 -4591.537,E2 -4591.537} C_VEL
LIN {X 0,Y 524.402,Z 601.5,A -85,B 0,C 180,E1 -4592.881,E2 -4592.881} C_VEL
LIN {X 0,Y 524.85,Z 591.394,A -85,B 0,C 180,E1 -4594.224,E2 -4594.224} C_VEL
LIN {X 0,Y 525.246,Z 581.049,A -85,B 0,C 180,E1 -4595.375,E2 -4595.375} C_VEL
LIN {X 0,Y 525.663,Z 569.79,A -85,B 0,C 180,E1 -4596.429,E2 -4596.429} C_VEL
LIN {X 0,Y 526.197,Z 557.497,A -85,B 0,C 180,E1 -4597.386,E2 -4597.386} C_VEL
LIN {X 0,Y 526.702,Z 543.995,A -85,B 0,C 180,E1 -4598.247,E2 -4598.247} C_VEL
LIN {X 0,Y 527.065,Z 531.014,A -85,B 0,C 180,E1 -4598.916,E2 -4598.916} C_VEL
LIN {X 0,Y 527.418,Z 516.857,A -85,B 0,C 180,E1 -4599.484,E2 -4599.484} C_VEL
LIN {X 0,Y 527.618,Z 502.116,A -85,B 0,C 180,E1 -4599.918,E2 -4599.918} C_VEL
LIN {X 0,Y 527.734,Z 486.564,A -85,B 0,C 180,E1 -4600.212,E2 -4600.212} C_VEL
LIN {X 0,Y 528.344,Z 376.561,A -85,B 0,C 180,E1 -4601.757,E2 -4601.757} C_VEL
LIN {X 0,Y 524.121,Z 366.635,A -85,B 0,C 180,E1 -4602.084,E2 -4602.084} C_VEL
LIN {X 0,Y 523.976,Z 365.842,A -85,B 0,C 180,E1 -4602.106,E2 -4602.106} C_VEL
LIN {X 0,Y 523.92,Z 365.852,A -85,B 0,C 180,E1 -4605.021,E2 -4605.021} C_VEL
LIN {X 0,Y 523.912,Z 365.845,A -85,B 0,C 180,E1 -4607.971,E2 -4607.971} C_VEL
LIN {X 0,Y 523.923,Z 365.845,A -85,B 0,C 180,E1 -4610.412,E2 -4610.412} C_VEL
LIN {X 0,Y 523.883,Z 365.856,A -85,B 0,C 180,E1 -4612.895,E2 -4612.895} C_VEL
LIN {X 0,Y 523.873,Z 365.854,A -85,B 0,C 180,E1 -4615.422,E2 -4615.422} C_VEL
LIN {X 0,Y 523.895,Z 365.848,A -85,B 0,C 180,E1 -4618.003,E2 -4618.003} C_VEL
LIN {X 0,Y 523.896,Z 365.846,A -85,B 0,C 180,E1 -4620.845,E2 -4620.845} C_VEL
LIN {X 0,Y 523.91,Z 365.845,A -85,B 0,C 180,E1 -4623.726,E2 -4623.726} C_VEL
LIN {X 0,Y 523.857,Z 365.852,A -85,B 0,C 180,E1 -4626.394,E2 -4626.394} C_VEL
LIN {X 0,Y 523.892,Z 365.856,A -85,B 0,C 180,E1 -4629.087,E2 -4629.087} C_VEL
LIN {X 0,Y 523.883,Z 365.848,A -85,B 0,C 180,E1 -4632.125,E2 -4632.125} C_VEL
LIN {X 0,Y 523.927,Z 365.85,A -85,B 0,C 180,E1 -4635.311,E2 -4635.311} C_VEL
LIN {X 0,Y 523.907,Z 365.846,A -85,B 0,C 180,E1 -4638.695,E2 -4638.695} C_VEL
LIN {X 0,Y 523.891,Z 365.854,A -85,B 0,C 180,E1 -4641.083,E2 -4641.083} C_VEL
LIN {X 0,Y 523.866,Z 365.852,A -85,B 0,C 180,E1 -4643.822,E2 -4643.822} C_VEL
LIN {X 0,Y 523.889,Z 365.846,A -85,B 0,C 180,E1 -4646.631,E2 -4646.631} C_VEL
LIN {X 0,Y 523.898,Z 365.854,A -85,B 0,C 180,E1 -4649.352,E2 -4649.352} C_VEL
LIN {X 0,Y 523.903,Z 365.845,A -85,B 0,C 180,E1 -4652.295,E2 -4652.295} C_VEL
LIN {X 0,Y 523.885,Z 365.853,A -85,B 0,C 180,E1 -4655.426,E2 -4655.426} C_VEL
LIN {X 0,Y 523.928,Z 365.844,A -85,B 0,C 180,E1 -4657.939,E2 -4657.939} C_VEL
LIN {X 0,Y 523.946,Z 365.838,A -85,B 0,C 180,E1 -4660.407,E2 -4660.407} C_VEL
LIN {X 0,Y 523.921,Z 365.844,A -85,B 0,C 180,E1 -4662.835,E2 -4662.835} C_VEL
LIN {X 0,Y 523.953,Z 365.845,A -85,B 0,C 180,E1 -4665.235,E2 -4665.235} C_VEL
LIN {X 0,Y 524.004,Z 365.821,A -85,B 0,C 180,E1 -4668.394,E2 -4668.394} C_VEL
LIN {X 0,Y 523.933,Z 365.843,A -85,B 0,C 180,E1 -4671.515,E2 -4671.515} C_VEL
LIN {X 0,Y 524.022,Z 365.83,A -85,B 0,C 180,E1 -4674.613,E2 -4674.613} C_VEL
LIN {X 0,Y 524.085,Z 365.826,A -85,B 0,C 180,E1 -4677.694,E2 -4677.694} C_VEL
LIN {X 0,Y 524.076,Z 365.826,A -85,B 0,C 180,E1 -4680,E2 -4680} C_VEL
LIN {X 0,Y 524.018,Z 365.832,A -85,B 0,C 180,E1 -4683.075,E2 -4683.075} C_VEL
LIN {X 0,Y 523.982,Z 365.837,A -85,B 0,C 180,E1 -4686.16,E2 -4686.16} C_VEL
LIN {X 0,Y 523.93,Z 365.844,A -85,B 0,C 180,E1 -4689.263,E2 -4689.263} C_VEL
LIN {X 0,Y 523.984,Z 365.843,A -85,B 0,C 180,E1 -4691.734,E2 -4691.734} C_VEL
LIN {X 0,Y 523.972,Z 365.836,A -85,B 0,C 180,E1 -4695.047,E2 -4695.047} C_VEL
LIN {X 0,Y 523.899,Z 365.848,A -85,B 0,C 180,E1 -4697.971,E2 -4697.971} C_VEL
LIN {X 0,Y 523.905,Z 365.846,A -85,B 0,C 180,E1 -4700.413,E2 -4700.413} C_VEL
LIN {X 0,Y 523.876,Z 365.847,A -85,B 0,C 180,E1 -4702.895,E2 -4702.895} C_VEL
LIN {X 0,Y 523.888,Z 365.852,A -85,B 0,C 180,E1 -4705.422,E2 -4705.422} C_VEL
LIN {X 0,Y 523.886,Z 365.853,A -85,B 0,C 180,E1 -4708.004,E2 -4708.004} C_VEL
LIN {X 0,Y 523.898,Z 365.847,A -85,B 0,C 180,E1 -4710.848,E2 -4710.848} C_VEL
LIN {X 0,Y 523.917,Z 365.847,A -85,B 0,C 180,E1 -4713.729,E2 -4713.729} C_VEL
LIN {X 0,Y 523.851,Z 365.854,A -85,B 0,C 180,E1 -4716.395,E2 -4716.395} C_VEL
LIN {X 0,Y 523.891,Z 365.845,A -85,B 0,C 180,E1 -4719.087,E2 -4719.087} C_VEL
LIN {X 0,Y 523.881,Z 365.852,A -85,B 0,C 180,E1 -4722.126,E2 -4722.126} C_VEL
LIN {X 0,Y 523.925,Z 365.845,A -85,B 0,C 180,E1 -4725.312,E2 -4725.312} C_VEL
LIN {X 0,Y 523.874,Z 365.845,A -85,B 0,C 180,E1 -4728.7,E2 -4728.7} C_VEL
LIN {X 0,Y 523.893,Z 365.855,A -85,B 0,C 180,E1 -4731.897,E2 -4731.897} C_VEL
LIN {X 0,Y 523.909,Z 365.847,A -85,B 0,C 180,E1 -4734.914,E2 -4734.914} C_VEL
LIN {X 0,Y 523.965,Z 365.974,A -85,B 0,C 180,E1 -4737.628,E2 -4737.628} C_VEL
LIN {X 0,Y 528.128,Z 381.719,A -85,B 0,C 180,E1 -4739.52,E2 -4739.52} C_VEL
LIN {X 0,Y 527.674,Z 404.139,A -85,B 0,C 180,E1 -4741.848,E2 -4741.848} C_VEL
LIN {X 0,Y 526.99,Z 432.537,A -85,B 0,C 180,E1 -4744.739,E2 -4744.739} C_VEL
LIN {X 0,Y 526.306,Z 463.588,A -85,B 0,C 180,E1 -4747.838,E2 -4747.838} C_VEL
LIN {X 0,Y 526.174,Z 470.376,A -85,B 0,C 180,E1 -4748.504,E2 -4748.504} C_VEL
LIN {X 0,Y 528.505,Z 485.457,A -85,B 0,C 180,E1 -4748.813,E2 -4748.813} C_VEL
LIN {X 0,Y 527.49,Z 639.711,A -85,B 0,C 180,E1 -4750.975,E2 -4750.975} C_VEL
LIN {X 0,Y 527.181,Z 655.705,A -85,B 0,C 180,E1 -4751.365,E2 -4751.365} C_VEL
LIN {X 0,Y 526.82,Z 670.455,A -85,B 0,C 180,E1 -4751.881,E2 -4751.881} C_VEL
LIN {X 0,Y 526.395,Z 684.419,A -85,B 0,C 180,E1 -4752.518,E2 -4752.518} C_VEL
LIN {X 0,Y 525.895,Z 698.144,A -85,B 0,C 180,E1 -4753.302,E2 -4753.302} C_VEL
LIN {X 0,Y 525.466,Z 711.777,A -85,B 0,C 180,E1 -4754.256,E2 -4754.256} C_VEL
LIN {X 0,Y 524.963,Z 724.886,A -85,B 0,C 180,E1 -4755.363,E2 -4755.363} C_VEL
LIN {X 0,Y 524.576,Z 737.4,A -85,B 0,C 180,E1 -4756.638,E2 -4756.638} C_VEL
LIN {X 0,Y 524.226,Z 746.874,A -85,B 0,C 180,E1 -4757.81,E2 -4757.81} C_VEL
LIN {X 0,Y 523.99,Z 756.083,A -85,B 0,C 180,E1 -4759.177,E2 -4759.177} C_VEL
LIN {X 0,Y 523.696,Z 763.741,A -85,B 0,C 180,E1 -4760.538,E2 -4760.538} C_VEL
LIN {X 0,Y 523.564,Z 770.088,A -85,B 0,C 180,E1 -4761.897,E2 -4761.897} C_VEL
LIN {X 0,Y 523.465,Z 775.999,A -85,B 0,C 180,E1 -4763.472,E2 -4763.472} C_VEL
LIN {X 0,Y 523.441,Z 779.385,A -85,B 0,C 180,E1 -4764.607,E2 -4764.607} C_VEL
LIN {X 0,Y 523.402,Z 782.886,A -85,B 0,C 180,E1 -4766.15,E2 -4766.15} C_VEL
LIN {X 0,Y 523.331,Z 785.189,A -85,B 0,C 180,E1 -4767.691,E2 -4767.691} C_VEL
LIN {X 0,Y 523.247,Z 786.347,A -85,B 0,C 180,E1 -4769.23,E2 -4769.23} C_VEL
LIN {X 0,Y 523.247,Z 786.347,A -85,B 0,C 180,E1 -4770.769,E2 -4770.769} C_VEL
LIN {X 0,Y 523.331,Z 785.186,A -85,B 0,C 180,E1 -4772.309,E2 -4772.309} C_VEL
LIN {X 0,Y 523.402,Z 782.883,A -85,B 0,C 180,E1 -4773.849,E2 -4773.849} C_VEL
LIN {X 0,Y 523.441,Z 779.388,A -85,B 0,C 180,E1 -4775.393,E2 -4775.393} C_VEL
LIN {X 0,Y 523.48,Z 774.611,A -85,B 0,C 180,E1 -4776.94,E2 -4776.94} C_VEL
LIN {X 0,Y 523.611,Z 768.422,A -85,B 0,C 180,E1 -4778.49,E2 -4778.49} C_VEL
LIN {X 0,Y 523.775,Z 760.645,A -85,B 0,C 180,E1 -4780.045,E2 -4780.045} C_VEL
LIN {X 0,Y 524.017,Z 752.37,A -85,B 0,C 180,E1 -4781.409,E2 -4781.409} C_VEL
LIN {X 0,Y 524.379,Z 742.371,A -85,B 0,C 180,E1 -4782.775,E2 -4782.775} C_VEL
LIN {X 0,Y 524.746,Z 731.924,A -85,B 0,C 180,E1 -4783.949,E2 -4783.949} C_VEL
LIN {X 0,Y 525.165,Z 719.397,A -85,B 0,C 180,E1 -4785.126,E2 -4785.126} C_VEL
LIN {X 0,Y 525.609,Z 706.869,A -85,B 0,C 180,E1 -4786.107,E2 -4786.107} C_VEL
LIN {X 0,Y 526.069,Z 693.267,A -85,B 0,C 180,E1 -4786.991,E2 -4786.991} C_VEL
LIN {X 0,Y 526.532,Z 678.304,A -85,B 0,C 180,E1 -4787.777,E2 -4787.777} C_VEL
LIN {X 0,Y 526.983,Z 662.549,A -85,B 0,C 180,E1 -4788.415,E2 -4788.415} C_VEL
